DATA_BLOCK "DOOR_EXTRACTOR_DB"	// DB 12
AUTHOR : Kamillas
VERSION : 0.1
  STRUCT
   DOOR_EXT_LOC_SS : BOOL ;	//DOOR EXTRACTOR LOCAL SELECTOR SWITCH
   DOOR_EXT_MAN_SS : BOOL ;	//DOOR EXTRACTOR MANUAL SELECTOR SWITCH
   DOOR_EXT_AUTO_SS : BOOL ;	//DOOR EXTRACTOR AUTO SELECTOR SWITCH
   DOOR_EXT_STP_PB : BOOL ;	//DOOR EXTRACTOR STOP PUSH BUTTON
   SLEW_FWD_STA_PB : BOOL ;	//SLEW FORWARD START PUSH BUTTON
   SLEW_RET_STA_PB : BOOL ;	//SLEW RETRACT START
   VER_COMP_FWD_STA_PB : BOOL ;	//VERTICAL COMPENSATION FORWARD START PUSH BUTTON
   VER_COMP_RET_STA_PB : BOOL ;	//VERTICAL COMPENSATION RETRACT START PUSH BUTTON
   TRA_FWD_STA_PB : BOOL ;	//TRAVEL FORWARD START PUSH BUTTON
   TRA_RET_STA_PB : BOOL ;	//TRAVEL RETRACT START PUSH BUTTON
   MAIN_STK_UP_STA_PB : BOOL ;	//MAIN STROKE UP START PUSH BUTTON
   MAIN_STK_UP_DN_PB : BOOL ;	//MAIN STROKE DOWN START PUSH BUTTON
   FIN_STK_UP_STA_PB : BOOL ;	//FINAL STROKE UP START PUSH BUTTON
   FIN_STK_UP_DN_PB : BOOL ;	//FINAL STROKE DOWN START PUSH BUTTON
   PRE_STK_UP_STA_PB : BOOL ;	//PRE STROKE UP START PUSH BUTTON
   PRE_STK_UP_DN_PB : BOOL ;	//PRE STROKE DOWN START PUSH BUTTON
   DR_SPNG_LK_STA_PB : BOOL ;	//DOOR SPRING PRESSURE START PUSH BUTTON
   DR_SPNG_UNLK_STA_PB : BOOL ;	//DOOR SPRING PRESSURE RELEASE START PUSH BUTTON
   DR_LCH_TURN_UP_PB : BOOL ;	//DOOR LATCH TURNING LOCK PUSH BUTTON
   DR_LCH_TURN_DN_PB : BOOL ;	//DOOR LATCH TURNING UNLOCK PUSH BUTTON
   EMERGENCY_PB_LCS_73 : BOOL ;	//EMERGENCY PUSHBUTTON LCS-73
   SLEW_FWD_STA_PB_LCS : BOOL ;	//SLEW FORWARD START PUSH BUTTON LCS
   SLEW_RET_STA_PB_LCS : BOOL ;	//SLEW RETRACT START PUSHBUTTON LCS
   VER_COMP_FWD_STA_PB_LCS : BOOL ;	//VERTICAL COMPENSATION FORWARD START LCS PUSH BUTTON
   VER_COMP_RET_STA_PB_LCS : BOOL ;	//VERTICAL COMPENSATION RETRACT START LCS PUSH BUTTON
   TRA_FWD_STA_PB_LCS : BOOL ;	//TRAVEL FORWARD START LCS  PUSH BUTTON
   TRA_RET_STA_PB_LCS : BOOL ;	//TRAVEL BACK START LCS  PUSH BUTTON
   MAIN_STK_UP_STA_PB_LCS : BOOL ;	//MAIN STROKE UP START LCS PUSH BUTTON
   MAIN_STK_DN_STA_PB_LCS : BOOL ;	//MAIN STROKE DN START LCS PUSH BUTTON
   FIN_STK_UP_STA_PB_LCS : BOOL ;	//FINAL STROKE UP START LCS  PUSH BUTTON
   FIN_STK_DN_STA_PB_LCS : BOOL ;	//FINAL STROKE DOWN START LCS PUSH BUTTON
   PRE_STK_UP_STA_PB_LCS : BOOL ;	//PREE STROKE UP START LCS PUSH BUTTON
   PRE_STK_DN_STA_PB_LCS : BOOL ;	//PREE STROKE DN START LCS PUSH BUTTON
   DR_SPNG_LK_STA_PB_LCS : BOOL ;	//DOOR SPRING LOCK START PUSH BUTTON LCS
   DR_SPNG_UNLK_STA_PB_LCS : BOOL ;	//DOOR SPRING UNLOCK  START PUSH BUTTON LCS
   LAMP_TEST_PB_LCS_73 : BOOL ;	//LAMP TEST PUSHBUTTON LCS-73
   DR_LCH_TURN_UP_PB_LCS : BOOL ;	//DOOR LATCH LOCK PUSH BUTTON LCS
   DR_LCH_TURN_DN_PB_LCS : BOOL ;	//DOOR LATCH UNLOCK PUSH BUTTON LCS
   DR_LCH_TURN_HOME_PB_LCS : BOOL ;	//DOOR LATCH HOME PUSH BUTTON LCS
   SLEW_SLOW_FWD_LS : BOOL ;	//SLEW SLOW FORWARD LIMIT SWITCH
   SLEW_SLOW_RET_LS : BOOL ;	//SLEW SLOW RETRACT LIMIT SWITCH
   SLEW_NOR_FWD_LS : BOOL ;	//SLEW NORMAL FORWARD LIMIT SWITCH
   SLEW_NOR_RET_LS : BOOL ;	//SLEW NORMAL RETRACT LIMIT SWITCH
   TRA_SLOW_FWD_LS : BOOL ;	//TRAVEL SLOW FORWARD LIMIT  SWITCH
   TRA_SLOW_RET_LS : BOOL ;	//TRAVEL SLOW RETRACT LIMIT  SWITCH
   TRA_FWD_LS : BOOL ;	//TRAVEL FORWARD LIMIT SWIITCH
   TRA_RET_LS : BOOL ;	//TRAVEL RETRACT LIMIT SWIITCH
   FOR_LS_TRAVEL : BOOL ;	//FORWARD LIMIT SWITCH TRAVEL
   DOOR_ON_HOOK_LS : BOOL ;	//DOOR ON HOOK LIMITSWTCH
   DOOR_FIX_LOC_FB_PR_SWT : BOOL ;	//DOOR FIX LOCKED FEEDBACK PRESSURE SWITCH
   DR_LCH_TURN_UP_LS : BOOL ;	//DOOR LATCH TURNING UP LIMIT SWICH
   DR_LCH_TURN_DN_LS : BOOL ;	//DOOR LATCH TURNING DOWN LIMIT SWICH
   SPRING_PRESS : BOOL ;	//SPRING PRESS
   SLEW_SLOW_FWD_CMD : BOOL ;	//SLEW SLOW FORWARD COMMAND
   SLEW_SLOW_RET_CMD : BOOL ;	//SLEW SLOW RETRACT COMMAND
   SLEW_NOR_FWD_COMMAND : BOOL ;	//SLEW NORMAL FORWARD COMMAND
   SLEW_NOR_RET_COMMAND : BOOL ;	//SLEW NORMAL RETRACT COMMAND
   VER_COMP_FWD_CMD : BOOL ;	//VERTICAL COMPENSATION FORWARD COMMAND
   VER_COMP_RET_CMD : BOOL ;	//VERTICAL COMPENSATION RETRACT COMMAND
   VER_COMP_RELIVE_CMD : BOOL ;	//VERTICAL COMPENSTAION RELIVE  COOMMAND
   TRA_SLOW_FWD_CMD : BOOL ;	//TRAVEL SLOW FORWARD COMMAND
   TRA_SLOW_RET_CMD : BOOL ;	//TRAVEL SLOW RETRACT COMMAND
   TRA_NOR_FWD_CMD : BOOL ;	//TRAVEL NORMAL FORWARD COMMAND
   TRA_NOR_RET_CMD : BOOL ;	//TRAVEL NORMAL RETRACT COMMAND
   TRA_RELIVE_CMD : BOOL ;	//TRAVEL RELIVE COOMMAND
   MAIN_STK_UP_CMD : BOOL ;	//MANUAL STROKE UP COMMAND
   MAIN_STK_DN_CMD : BOOL ;	//MANUAL STROKE DN COMMAND
   PRE_STK_UP_CMD : BOOL ;	//PRE STROKE UP COMMAND
   PRE_STK_DN_CMD : BOOL ;	//PRE STROKE DN COMMAND
   DR_SPNG_LK_CMD : BOOL ;	//DOOR SPRING PRESS LOCK COMMAND
   DR_SPNG_UNLK_CMD : BOOL ;	//DOOR SPRING PRESS UNLOCK COMMAND
   DR_LCH_TURN_UP_CMD : BOOL ;	//DOOR LATCH TURNING UP COMMAND
   DR_LCH_TURN_DN_CMD : BOOL ;	//DOOR LATCH TURNING DOWN COMMADN
   SLEW_SLOW_FWD_IND : BOOL ;	//SLEW SLOW FORWARD INDICATOR
   SLEW_SLOW_RET_IND : BOOL ;	//SLEW SLOW RETRACT INDICATOR
   VER_COMP_FWD_IND : BOOL ;	//VERTICAL COMPENSATION FORWARD INDICATOR
   VER_COMP_RET_IND : BOOL ;	//VERTICAL COMPENSATION RETRACT INDICATOR
   TRA_FWD_IND : BOOL ;	//TRAVEL FORWARD INDICATOR
   TRA_RET_IND : BOOL ;	//TRAVEL BACK INDICATOR
   MAIN_STK_UP_IND : BOOL ;	//FINAL STROKE  UP INDICATION
   MAIN_STK_DN_IND : BOOL ;	//FINAL STROKE  DOWN  INDICATOR
   FIN_STK_UP_IND : BOOL ;	//FINAL STROKE  UP INDICATOR
   FIN_STK_DN_IND : BOOL ;	//FINAL STROKE  DOWN INDICATOR
   PRE_STK_UP_IND : BOOL ;	//PRE STROKE  UP INDICATION
   PRE_STK_DN_IND : BOOL ;	//PRE STROKE  DOWN INDICATOR
   DR_SPNG_LK_IND : BOOL ;	//DOOR SPRING PRESS LOCK INDICATOR
   DR_SPNG_UNLK_IND : BOOL ;	//DOOR SPRING PRESS UNLOCK INDICATOR
   DOOR_FIX_LOCK_IND : BOOL ;	//DOOR FIX LOCK INDICATOR
   DOOR_FIX_UNLK_IND : BOOL ;	//DOOR FIX UNLOCK INDICATOR
   DOOR_FIX_UNLK_IND1 : BOOL ;	//DOOR FIX UNLOCK INDICATOR
   LCS_73_ON_IND : BOOL ;	//LCS-73_ON_INDICATOR
   SLEW_SLOW_FWD_IND_LCS : BOOL ;	//SLEW SLOW FORWARD INDICATOR LCS
   SLEW_SLOW_RET_IND_LCS : BOOL ;	//SLEW SLOW RETRACT INDICATOR LCS
   VER_COMP_FWD_IND_LCS : BOOL ;	//VERTICAL COMPENSATION FORWARD INDICATOR LCS
   VER_COMP_RET_IND_LCS : BOOL ;	//VERTICAL COMPENSATION RETRACT INDICATOR LCS
   TRA_FWD_IND_LCS : BOOL ;	//TRAVEL FORWARD INDICATOR
   TRA_RET_IND_LCS : BOOL ;	//TRAVEL BACK INDICATOR LCS
   MAIN_STK_UP_IND_LCS : BOOL ;	//FINAL STROKE UP INDICATION LCS
   MAIN_STK_DN_IND_LCS : BOOL ;	//FINAL STROKE DOWN  INDICATOR LCS
   FIN_STK_UP_IND_LCS : BOOL ;	//FINAL STROKE UP INDICATOR LCS
   FIN_STK_DN_IND_LCS : BOOL ;	//FINAL STROKE DOWN INDICATOR LCS
   PRE_STK_UP_IND_LCS : BOOL ;	//PRE STROKE UP INDICATION LCS
   PRE_STK_DN_IND_LCS : BOOL ;	//PRE STROKE DOWN INDICATOR LCS
   DR_LCH_TURN_HOME_IND_LCS : BOOL ;	//DOOR LATCH HOME INDICATION LCS
   DR_LCH_TURN_UP_IND_LCS : BOOL ;	//DOOR LATCH TURNING UP INDICATOR LCS
   DR_LCH_TURN_DN_IND_LCS : BOOL ;	//DOOR LATCH TURNING DOWN INDICATOR LCS
   DOOR_FIX_LOCK_IND_LCS : BOOL ;	//DOOR FIX LOCK INDICATOR LCS
   DOOR_FIX_UNLK_IND_LCS : BOOL ;	//DOOR FIX UNLOCK INDICATOR LCS
   SLEW_SL_FWD_OP_CUT : BOOL ;	//SLEW SLOW FORWARD OUTPUT CUT
   SLEW_SL_FWD_FLT_TMR : INT ;	//SLEW SLOW FORWARD FAULT TIMER
   SLEW_SL_FWD_FLT_GEN : INT  := 8;	//SLEW SLOW FORWARD FAULT GENERATION TIME
   SLEW_SL_FWD_OP_CT_TM : INT ;	//SLEW SLOW FORWARD OUTPUT CUT TIMER
   SLEW_SL_FWD_FLT : BOOL ;	//SLEW SLOW FORWARD FAULT
   SLEW_SL_AUTO_FWD_OVR : BOOL ;	//SLEW SLOW AUTO FORWARD OVER
   SLEW_SL_AUTO_FWD_DEL : INT  := 3;	//SLEW SLOW AUTO FORWARD OVER DELAY
   SLEW_SL_ATO_FWD_DL_T : INT ;	//SLEW SLOW AUTO FORWARD OVER DELAY TIMER
   SLEW_NR_FWD_OP_CUT : BOOL ;	//SLEW NORMAL FORWARD OUTPUT CUT
   SLEW_NR_FWD_FLT_TMR : INT ;	//SLEW NORMAL FORWARD FAULT TIMER
   SLEW_NR_FWD_FLT_GEN : INT  := 8;	//SLEW NORMAL FORWARD FAULT GENERATION TIME
   SLEW_NR_FWD_OP_CT_TM : INT ;	//SLEW NORMAL FORWARD OUTPUT CUT TIMER
   SLEW_NR_FWD_FLT : BOOL ;	//SLEW NORMAL FORWARD FAULT
   SLEW_NR_AUTO_FWD_OVR : BOOL ;	//SLEW NORMAL AUTO FORWARD OVER
   SLEW_NR_AUTO_FWD_DEL : INT  := 3;	//SLEW NORMAL AUTO FORWARD OVER DELAY
   SLEW_NR_ATO_FWD_DL_T : INT ;	//SLEW NORMAL AUTO FORWARD OVER DELAY TIMER
   PULSE_1 : BOOL ;	//PULSE 1
   PULSE_2 : BOOL ;	//PULSE 2
   PULSE_3 : BOOL ;	//PULSE 3
   PULSE_4 : BOOL ;	//PULSE 4
   PULSE_5 : BOOL ;	//PULSE 5
   PULSE_6 : BOOL ;	//PULSE 6
   PULSE_7 : BOOL ;	//PULSE 7
   PULSE_8 : BOOL ;	//PULSE 8
   PULSE_9 : BOOL ;	//PULSE 9
   PULSE_10 : BOOL ;	//PULSE 10
   PULSE_11 : BOOL ;	//PULSE 11
   PULSE_12 : BOOL ;	//PULSE 12
   PULSE_13 : BOOL ;	//PULSE 13
   PULSE_14 : BOOL ;	//PULSE 14
   PULSE_15 : BOOL ;	//PULSE 15
   PULSE_16 : BOOL ;	//PULSE 16
   SLEW_NR_RET_OP_CUT : BOOL ;	//SLEW NORMAL RETRACT OUTPUT CUT
   SLEW_NR_RET_FLT_TMR : INT ;	//SLEW NORMAL RETRACT FAULT TIMER
   SLEW_NR_RET_FLT_GEN : INT  := 8;	//SLEW NORMAL RETRACT FAULT GENERATION TIME
   SLEW_NR_RET_OP_CT_TM : INT ;	//SLEW NORMAL RETRACT RETRACT OUTPUT CUT TIMER
   SLEW_NR_RET_FLT : BOOL ;	//SLEW NORMAL RETRACT RETRACT FAULT
   SLEW_NR_AUTO_RET_OVR : BOOL ;	//SLEW NORMAL AUTO RETRACT OVER
   SLEW_NR_AUTO_RET_DEL : INT  := 3;	//SLEW NORMAL AUTO RETRACT OVER DELAY
   SLEW_NR_ATO_RET_DL_T : INT ;	//SLEW NORMAL AUTO RETRACT OVER DELAY TIMER
   VER_COMP_FWD_OP_CUT : BOOL ;	//VERTICAL COMPENSATION FORWARD OUTPUT CUT
   VER_COMP_FWD_FLT_TMR : INT ;	//VERTICAL COMPENSATION FORWARD FAULT TIMER
   VER_COMP_FWD_FLT_GEN : INT  := 8;	//VERTICAL COMPENSATION FORWARD FAULT GENERATION TIME
   VER_COMP_FWD_OP_CT_TM : INT ;	//VERTICAL COMPENSATION FORWARD OUTPUT CUT TIMER
   VER_COMP_FWD_FLT : BOOL ;	//VERTICAL COMPENSATION FORWARD FAULT
   VER_COMP_AUTO_FWD_OVR : BOOL ;	//VERTICAL COMPENSATION AUTO FORWARD OVER
   VER_COMP_AUTO_FWD_DEL : INT  := 3;	//VERTICAL COMPENSATION AUTO FORWARD OVER DELAY
   VER_COMP_ATO_FWD_DL_T : INT ;	//VERTICAL COMPENSATION AUTO FORWARD OVER DELAY TIMER
   VER_COMP_RET_OP_CUT : BOOL ;	//VERTICAL COMPENSATION RETRACT OUTPUT CUT
   VER_COMP_RET_FLT_TMR : INT ;	//VERTICAL COMPENSATION RETRACT FAULT TIMER
   VER_COMP_RET_FLT_GEN : INT  := 8;	//VERTICAL COMPENSATION RETRACT FAULT GENERATION TIME
   VER_COMP_RET_OP_CT_TM : INT ;	//VERTICAL COMPENSATION RETRACT OUTPUT CUT TIMER
   VER_COMP_RET_FLT : BOOL ;	//VERTICAL COMPENSATION RETRACT FAULT
   VER_COMP_AUTO_RET_OVR : BOOL ;	//VERTICAL COMPENSATION AUTO RETRACT OVER
   VER_COMP_AUTO_RET_DEL : INT  := 3;	//VERTICAL COMPENSATION AUTO RETRACT OVER DELAY
   VER_COMP_ATO_RET_DL_T : INT ;	//VERTICAL COMPENSATION AUTO RETRACT OVER DELAY TIMER
   TRA_SLOW_FWD_OP_CUT : BOOL ;	//TRAVEL SLOW FORWARD OUTPUT CUT
   TRA_SLOW_FWD_FLT_TMR : INT ;	//TRAVEL SLOW FORWARD FAULT TIMER
   TRA_SLOW_FWD_FLT_GEN : INT  := 8;	//TRAVEL SLOW FORWARD FAULT GENERATION TIME
   TRA_SLOW_FWD_OP_CT_TM : INT ;	//TRAVEL SLOW FORWARD OUTPUT CUT TIMER
   TRA_SLOW_FWD_FLT : BOOL ;	//TRAVEL SLOW FORWARD FAULT
   TRA_SLOW_AUTO_FWD_OVR : BOOL ;	//TRAVEL SLOW AUTO FORWARD OVER
   TRA_SLOW_AUTO_FWD_DEL : INT  := 3;	//TRAVEL SLOW AUTO FORWARD OVER DELAY
   TRA_SLOW_ATO_FWD_DL_T : INT ;	//TRAVEL SLOW AUTO FORWARD OVER DELAY TIMER
   TRA_SLOW_RET_OP_CUT : BOOL ;	//TRAVEL SLOW RETRACT OUTPUT CUT
   TRA_SLOW_RET_FLT_TMR : INT ;	//TRAVEL SLOW RETRACT FAULT TIMER
   TRA_SLOW_RET_FLT_GEN : INT  := 8;	//TRAVEL SLOW RETRACT FAULT GENERATION TIME
   TRA_SLOW_RET_OP_CT_TM : INT ;	//TRAVEL SLOW RETRACT OUTPUT CUT TIMER
   TRA_SLOW_RET_FLT : BOOL ;	//TRAVEL SLOW RETRACT FAULT
   TRA_SLOW_AUTO_RET_OVR : BOOL ;	//TRAVEL SLOW AUTO RETRACT OVER
   TRA_SLOW_AUTO_RET_DEL : INT  := 3;	//TRAVEL SLOW AUTO RETRACT OVER DELAY
   TRA_SLOW_ATO_RET_DL_T : INT ;	//TRAVEL SLOW AUTO RETRACT OVER DELAY TIMER
   TRA_NOR_FWD_OP_CUT : BOOL ;	//TRAVEL NORMAL FORWARD OUTPUT CUT
   TRA_NOR_FWD_FLT_TMR : INT ;	//TRAVEL NORMAL FORWARD FAULT TIMER
   TRA_NOR_FWD_FLT_GEN : INT  := 8;	//TRAVEL NORMAL FORWARD FAULT GENERATION TIME
   TRA_NOR_FWD_OP_CT_TM : INT ;	//TRAVEL NORMAL FORWARD OUTPUT CUT TIMER
   TRA_NOR_FWD_FLT : BOOL ;	//TRAVEL NORMAL FORWARD FAULT
   TRA_NOR_AUTO_FWD_OVR : BOOL ;	//TRAVEL NORMAL AUTO FORWARD OVER
   TRA_NOR_AUTO_FWD_DEL : INT  := 3;	//TRAVEL NORMAL AUTO FORWARD OVER DELAY
   TRA_NOR_ATO_FWD_DL_T : INT ;	//TRAVEL NORMAL AUTO FORWARD OVER DELAY TIMER
   TRA_NOR_RET_OP_CUT : BOOL ;	//TRAVEL NORMAL RETRACT OUTPUT CUT
   TRA_NOR_RET_FLT_TMR : INT ;	//TRAVEL NORMAL RETRACT FAULT TIMER
   TRA_NOR_RET_FLT_GEN : INT  := 8;	//TRAVEL NORMAL RETRACT FAULT GENERATION TIME
   TRA_NOR_RET_OP_CT_TM : INT ;	//TRAVEL NORMAL RETRACT OUTPUT CUT TIMER
   TRA_NOR_RET_FLT : BOOL ;	//TRAVEL NORMAL RETRACT FAULT
   TRA_NOR_AUTO_RET_OVR : BOOL ;	//TRAVEL NORMAL AUTO RETRACT OVER
   TRA_NOR_AUTO_RET_DEL : INT  := 3;	//TRAVEL NORMAL AUTO RETRACT OVER DELAY
   TRA_NOR_ATO_RET_DL_T : INT ;	//TRAVEL NORMAL AUTO RETRACT OVER DELAY TIMER
   MAIN_STK_UP_OP_CUT : BOOL ;	//MAIN STROK UP OUTPUT CUT
   MAIN_STK_UP_FLT_TMR : INT ;	//MAIN STROK UP FAULT TIMER
   MAIN_STK_UP_FLT_GEN : INT  := 8;	//MAIN STROK UP FAULT GENERATION TIME
   MAIN_STK_UP_OP_CT_TM : INT ;	//MAIN STROK UP OUTPUT CUT TIMER
   MAIN_STK_UP_FLT : BOOL ;	//MAIN STROK UP FAULT
   MAIN_STK_AUTO_UP_OVR : BOOL ;	//MAIN STROK AUTO UP OVER
   MAIN_STK_AUTO_UP_DEL : INT  := 3;	//MAIN STROK AUTO UP OVER DELAY
   MAIN_STK_ATO_UP_DL_T : INT ;	//MAIN STROK AUTO UP OVER DELAY TIMER
   MAIN_STK_DN_OP_CUT : BOOL ;	//MAIN STROK DOWN OUTPUT CUT
   MAIN_STK_DN_FLT_TMR : INT ;	//MAIN STROK DOWN FAULT TIMER
   MAIN_STK_DN_FLT_GEN : INT  := 8;	//MAIN STROK DOWN FAULT GENERATION TIME
   MAIN_STK_DN_OP_CT_TM : INT ;	//MAIN STROK DOWN OUTPUT CUT TIMER
   MAIN_STK_DN_FLT : BOOL ;	//MAIN STROK DOWN FAULT
   MAIN_STK_AUTO_DN_OVR : BOOL ;	//MAIN STROK AUTO DOWN OVER
   MAIN_STK_AUTO_DN_DEL : INT  := 3;	//MAIN STROK AUTO DOWN OVER DELAY
   MAIN_STK_ATO_DN_DL_T : INT ;	//MAIN STROK AUTO DOWN OVER DELAY TIMER
   PRE_STK_UP_OP_CUT : BOOL ;	//PRE STROK UP OUTPUT CUT
   PRE_STK_UP_FLT_TMR : INT ;	//PRE STROK UP FAULT TIMER
   PRE_STK_UP_FLT_GEN : INT  := 8;	//PRE STROK UP FAULT GENERATION TIME
   PRE_STK_UP_OP_CT_TM : INT ;	//PRE STROK UP OUTPUT CUT TIMER
   PRE_STK_UP_FLT : BOOL ;	//PRE STROK UP FAULT
   PRE_STK_AUTO_UP_OVR : BOOL ;	//PRE STROK AUTO UP OVER
   PRE_STK_AUTO_UP_DEL : INT  := 3;	//PRE STROK AUTO UP OVER DELAY
   PRE_STK_ATO_UP_DL_T : INT ;	//PRE STROK AUTO UP OVER DELAY TIMER
   PRE_STK_DN_OP_CUT : BOOL ;	//PRE STROK DOWN OUTPUT CUT
   PRE_STK_DN_FLT_TMR : INT ;	//PRE STROK DOWN FAULT TIMER
   PRE_STK_DN_FLT_GEN : INT  := 8;	//PRE STROK DOWN FAULT GENERATION TIME
   PRE_STK_DN_OP_CT_TM : INT ;	//PRE STROK DOWN OUTPUT CUT TIMER
   PRE_STK_DN_FLT : BOOL ;	//PRE STROK DOWN FAULT
   PRE_STK_AUTO_DN_OVR : BOOL ;	//PRE STROK AUTO DOWN OVER
   PRE_STK_AUTO_DN_DEL : INT  := 3;	//PRE STROK AUTO DOWN OVER DELAY
   PRE_STK_ATO_DN_DL_T : INT ;	//PRE STROK AUTO DOWN OVER DELAY TIMER
   FIN_STK_UP_OP_CUT : BOOL ;	//FINAL STROK UP OUTPUT CUT
   FIN_STK_UP_FLT_TMR : INT ;	//FINAL STROK UP FAULT TIMER
   FIN_STK_UP_FLT_GEN : INT  := 8;	//FINAL STROK UP FAULT GENERATION TIME
   FIN_STK_UP_OP_CT_TM : INT ;	//FINAL STROK UP OUTPUT CUT TIMER
   FIN_STK_UP_FLT : BOOL ;	//FINAL STROK UP FAULT
   FIN_STK_AUTO_UP_OVR : BOOL ;	//FINAL STROK AUTO UP OVER
   FIN_STK_AUTO_UP_DEL : INT  := 3;	//FINAL STROK AUTO UP OVER DELAY
   FIN_STK_ATO_UP_DL_T : INT ;	//FINAL STROK AUTO UP OVER DELAY TIMER
   FIN_STK_DN_OP_CUT : BOOL ;	//FINAL STROK DOWN OUTPUT CUT
   FIN_STK_DN_FLT_TMR : INT ;	//FINAL STROK DOWN FAULT TIMER
   FIN_STK_DN_FLT_GEN : INT  := 8;	//FINAL STROK DOWN FAULT GENERATION TIME
   FIN_STK_DN_OP_CT_TM : INT ;	//FINAL STROK DOWN OUTPUT CUT TIMER
   FIN_STK_DN_FLT : BOOL ;	//FINAL STROK DOWN FAULT
   FIN_STK_AUTO_DN_OVR : BOOL ;	//FINAL STROK AUTO DOWN OVER
   FIN_STK_AUTO_DN_DEL : INT  := 3;	//FINAL STROK AUTO DOWN OVER DELAY
   FIN_STK_ATO_DN_DL_T : INT ;	//FINAL STROK AUTO DOWN OVER DELAY TIMER
   FIN_STK_UP_CMD : BOOL ;	//FINAL STROKE UP COMMAND
   FIN_STK_DN_CMD : BOOL ;	//FINAL STROKE DOWN COMMAND
   DR_SPNG_LK_OP_CUT : BOOL ;	//DOOR SPRING PRESSURE LOCK OUTPUT CUT
   DR_SPNG_LK_FLT_TMR : INT ;	//DOOR SPRING PRESSURE LOCK FAULT TIMER
   DR_SPNG_LK_FLT_GEN : INT  := 8;	//DOOR SPRING PRESSURE LOCK FAULT GENERATION TIME
   DR_SPNG_LK_OP_CT_TM : INT ;	//DOOR SPRING PRESSURE LOCK OUTPUT CUT TIMER
   DR_SPNG_LK_FLT : BOOL ;	//DOOR SPRING PRESSURE LOCK FAULT
   DR_SPNG_AUTO_LK_OVR : BOOL ;	//DOOR SPRING AUTO PRESSURE LOCK OVER
   DR_SPNG_AUTO_LK_DEL : INT  := 3;	//DOOR SPRING AUTO PRESSURE LOCK OVER DELAY
   DR_SPNG_ATO_LK_DL_T : INT ;	//DOOR SPRING AUTO PRESSURE LOCK OVER DELAY TIMER
   DR_SPNG_UNLK_OP_CUT : BOOL ;	//DOOR SPRING PRESSURE UNLOCK OUTPUT CUT
   DR_SPNG_UNLK_FLT_TMR : INT ;	//DOOR SPRING PRESSURE UNLOCK FAULT TIMER
   DR_SPNG_UNLK_FLT_GEN : INT  := 8;	//DOOR SPRING PRESSURE UNLOCK FAULT GENERATION TIME
   DR_SPNG_UNLK_OP_CT_TM : INT ;	//DOOR SPRING PRESSURE UNLOCK OUTPUT CUT TIMER
   DR_SPNG_UNLK_FLT : BOOL ;	//DOOR SPRING PRESSURE UNLOCK FAULT
   DR_SPNG_AUTO_UNLK_OVR : BOOL ;	//DOOR SPRING AUTO PRESSURE UNLOCK OVER
   DR_SPNG_AUTO_UNLK_DEL : INT  := 3;	//DOOR SPRING AUTO PRESSURE UNLOCK OVER DELAY
   DR_SPNG_ATO_UNLK_DL_T : INT ;	//DOOR SPRING AUTO PRESSURE UNLOCK OVER DELAY TIMER
   PULSE_17 : BOOL ;	//PULSE 17
   PULSE_18 : BOOL ;	//PULSE 18
   PULSE_19 : BOOL ;	//PULSE 19
   PULSE_20 : BOOL ;	//PULSE 20
   PULSE_21 : BOOL ;	//PULSE 21
   PULSE_22 : BOOL ;	//PULSE 22
   PULSE_23 : BOOL ;	//PULSE 23
   PULSE_24 : BOOL ;	//PULSE 24
   PULSE_25 : BOOL ;	//PULSE 25
   PULSE_26 : BOOL ;	//PULSE 26
   PULSE_27 : BOOL ;	//PULSE 27
   PULSE_28 : BOOL ;	//PULSE 28
   PULSE_29 : BOOL ;	//PULSE 29
   PULSE_30 : BOOL ;	//PULSE 30
   DR_LCH_UP_OP_CUT : BOOL ;	//DOOR LATCH UP OUTPUT CUT
   DR_LCH_UP_FLT_TMR : INT ;	//DOOR LATCH UP FAULT TIMER
   DR_LCH_UP_FLT_GEN : INT  := 8;	//DOOR LATCH UP FAULT GENERATION TIME
   DR_LCH_UP_OP_CT_TM : INT ;	//DOOR LATCH UP OUTPUT CUT TIMER
   DR_LCH_UP_FLT : BOOL ;	//DOOR LATCH UP FAULT
   DR_LCH_AUTO_UP_OVR : BOOL ;	//DOOR LATCH AUTO PRESSURE UP OVER
   DR_LCH_AUTO_UP_DEL : INT  := 3;	//DOOR LATCH AUTO PRESSURE UP OVER DELAY
   DR_LCH_ATO_UP_DL_T : INT ;	//DOOR LATCH AUTO PRESSURE UP OVER DELAY TIMER
   DR_LCH_DN_OP_CUT : BOOL ;	//DOOR LATCH DOWN OUTPUT CUT
   DR_LCH_DN_FLT_TMR : INT ;	//DOOR LATCH DOWN FAULT TIMER
   DR_LCH_DN_FLT_GEN : INT  := 8;	//DOOR LATCH DOWN FAULT GENERATION TIME
   DR_LCH_DN_OP_CT_TM : INT ;	//DOOR LATCH DOWN OUTPUT CUT TIMER
   DR_LCH_DN_FLT : BOOL ;	//DOOR LATCH DOWN FAULT
   DR_LCH_AUTO_DN_OVR : BOOL ;	//DOOR SPRING AUTO PRESSURE DOWN OVER
   DR_LCH_AUTO_DN_DEL : INT  := 3;	//DOOR SPRING AUTO PRESSURE DOWN OVER DELAY
   DR_LCH_ATO_DN_DL_T : INT ;	//DOOR SPRING AUTO PRESSURE DOWN OVER DELAY TIMER
   TRA_SLOW_FWD_IND : BOOL ;	//TRAVEL SLOW FORWARD INDICATOR
   TRA_SLOW_RET_IND : BOOL ;	//TRAVEL SLOW RETRACT INDICATOR
   TRA_SLOW_FWD_IND_LCS : BOOL ;	//TRAVEL SLOW FORWARD INDICATOR LCS
   TRA_SLOW_RET_IND_LCS : BOOL ;	//TRAVEL RETRACT INDICATOR LCS
   SLEW_FWD_IND : BOOL ;	//SLEW NORMAL FORWARD INDICATOR
   SLEW_RET_IND : BOOL ;	//SLEW NORMAL RETRACT INDICATOR
   SLEW_FWD_IND_LCS : BOOL ;	//SLEW NORMAL FORWARD INDICATOR LCS
   SLEW_RET_IND_LCS : BOOL ;	//SLEW NORMAL RETRACT INDICATOR LCS
   DR_SPNG_LK_IND_LCS : BOOL ;	//DOOR SPRING PRESS LOCK INDICATOR LCS
   DR_SPNG_UNLK_IND_LCS : BOOL ;	//DOOR SPRING PRESS UNLOCK INDICATOR LCS
   DE_TRA_SLOW_FWD_BIT : BOOL ;	//DOOR EXTRACTOR TRAVEL SLOW FORWARD START BIT
   DOR_EXT_RPL_ILK_BIT : BOOL ;	//DOOR EXTRACTOR/REPLACE INTERLOCK BIT
   DR_EXT_AUTO_STA_BIT : BOOL ;	//DOOR EXTRACTOR AUTO START BIT
   EXT_OVEN_DOR_AUTO_STA_PB : BOOL ;	//EXTRACT OVEN DOOR AUTO START PUSH BUTTON
   DR_EXT_RPL_AUTO_STP_PB : BOOL ;	//DOOR EXTRACTOR/REPLACE AUTO STOP PUSH BUTTON
   RPL_OVEN_DOR_AUTO_STA_PB : BOOL ;	//REPLACE OVEN DOOR AUTO START PUSH BUTTON
   VER_COMP_LDT_SCLD_VLU : REAL ;	//VERTICAL COMPENSATION LDT SCALED VALUE
   VER_COMP_LDT_SLNG_ERR : WORD ;	//VERTICAL COMPENSATION LDT SCALING ERROR
   DR_RPL_AUTO_STA_BIT : BOOL ;	//DOOR REPLACE AUTO START BIT
   PULSE_31 : BOOL ;	//PULSE 31
   PULSE_32 : BOOL ;	//PULSE 32
   PULSE_33 : BOOL ;	//PULSE 33
   PULSE_34 : BOOL ;	//PULSE 34
   PULSE_35 : BOOL ;	//PULSE 35
   PULSE_36 : BOOL ;	//PULSE 36
   PULSE_37 : BOOL ;	//PULSE 37
   PULSE_38 : BOOL ;	//PULSE 38
   PULSE_39 : BOOL ;	//PULSE 39
   PULSE_40 : BOOL ;	//PULSE 40
   PULSE_41 : BOOL ;	//PULSE 41
   PULSE_42 : BOOL ;	//PULSE 42
   PULSE_43 : BOOL ;	//PULSE 43
   PULSE_44 : BOOL ;	//PULSE 44
   PULSE_45 : BOOL ;	//PULSE 45
   PULSE_46 : BOOL ;	//PULSE 46
   PULSE_47 : BOOL ;	//PULSE 47
   PULSE_48 : BOOL ;	//PULSE 48
   PULSE_49 : BOOL ;	//PULSE 49
   PULSE_50 : BOOL ;	//PULSE 50
   PRE_STK_UP_LR : BOOL ;	//PRE STROKE UP LIMIT READHED
   PRE_STK_DN_LR : BOOL ;	//PRE STROKE DOWN LIMIT READHED
   MAIN_STK_FWD_LR : BOOL ;	//MAIN STROKE UP LIMIT READHED
   MAIN_STK_DN_LR : BOOL ;	//MAIN STROKE DOWN LIMIT READHED
   FIN_STK_FWD_LR : BOOL ;	//FINAL STROKE UP LIMIT READHED
   FIN_STK_DN_LR : BOOL ;	//FINAL STROKE DOWN LIMIT READHED
   EXT_OVEN_DOR_IND : BOOL ;	//EEXTRACT OVEN DOOR INDICATOR
   RPL_OVEN_DOR_IND : BOOL ;	//REPLACE OVEN DOOR INDICATOR
   SLEW_AUTO_FWD_SET : BOOL ;	//SLWE AUTO FORWARD SET
   SLEW_AUTO_RET_SET : BOOL ;	//SLWE AUTO RETRACT SET
   VER_COMP_AUTO_FWD_SET : BOOL ;	//VERTICAL COMPENSATION AUTO FORWARD SET
   VER_COMP_AUTO_RET_SET : BOOL ;	//VERTICAL COMPENSATION AUTO RETRACT SET
   TRA_AUTO_FWD_SET : BOOL ;	//TRAVEL AUTO FORWARD SET
   TRA_AUTO_RET_SET : BOOL ;	//TRAVEL AUTO RETRACT SET
   PRE_STK_AUTO_FWD_SET : BOOL ;	//PRE STROK AUTO FORWARD SET
   PRE_STK_AUTO_RET_SET : BOOL ;	//PRE STROK AUTO RETRACT SET
   MAIN_STK_AUTO_FWD_SET : BOOL ;	//MAIN STROK AUTO FORWARD SET
   MAIN_STK_AUTO_RET_SET : BOOL ;	//MAIN STROK AUTO RETRACT SET
   FIN_STK_AUTO_FWD_SET : BOOL ;	//FINAL STROK AUTO FORWARD SET
   FIN_STK_AUTO_RET_SET : BOOL ;	//FINAL STROK AUTO RETRACT SET
   DR_SPNG_AUTO_PRSD_SET : BOOL ;	//DOOR SPING AUTO PRESSED SET
   DR_SRNG_AUTO_RLSD_SET : BOOL ;	//DOOR SPING AUTO RELESED SET
   DR_LCH_TURN_AUTO_UP_SET : BOOL ;	//DOOR LATCH TURN AUTO UP BIT
   DR_LCH_TURN_AUTO_DN_SET : BOOL ;	//DOOR LATCH TURN AUTO DOWN BIT
   DR_LFT_LDT_SCLD_VLU : REAL ;	//DOOR LIFTING LDT SCALED VALUE
   DR_LFT_LDT_SLNG_ERR : WORD ;	//DOOR LIFTING LDT SCALING ERROR
   VER_COMP_VALUE : REAL ;	//VERTICAL COMPENSATION VALUE
   VER_COMP_LDT_REAL : REAL ;	//VERTICAL COMPENSATION LDT REAL VALUE
   DR_LFT_LDT_REAL : REAL ;	//DOOR LIFTING LDT REAL VALUE
   VER_COMP_UNSCLD_VLU : INT ;	//VERTICAL COMPENSATION UNSCALED VALUE
   DR_LFT_UNSCLD_VLU : INT ;	//DOOR LIFTER UNSCALED VALUE
   PRE_STK_UP_LDT_VLU : REAL ;	//PRE STROKE UP LDT VALUE
   MAIN_STK_UP_LDT_VLU : REAL ;	//MAIN STROKE UP LDT VALUE
   FIN_STK_UP_LDT_VLU : REAL ;	//FIN STROKE UP LDT VALUE
   PRE_STK_DN_LDT_VLU : REAL ;	//PRE STROKE DOWN LDT VALUE
   MAIN_STK_DN_LDT_VLU : REAL ;	//MAIN STROKE DOWN LDT VALUE
   FIN_STK_DN_LDT_VLU : REAL ;	//FIN STROKE DOWN LDT VALUE
   VER_COMP_FWD_LIM_VALUE : REAL ;	//VERTICAL COMPENSATION FORWARD LIMIT VALUE
   DOOR_FIX_REL_FB : BOOL ;	//DOOR RELEASE FEEDBACK
   DR_LCH_TURN_UP_IND : BOOL ;	//DOOR LATCH LOCK INDICATOR CD
   DR_LCH_TURN_DN_IND : BOOL ;	//DOOR LATCH UNLOCK INDICATOR CD
   VER_COMP_LR : BOOL ;	//VERTICAL COMPENSATION LIMIT REACHED
   DR_EXTR_HME_POS : BOOL ;	//DOOR EXTRACTOR HOME POSITION REACHED
   DR_EXT_AUTO_OPER_FIN : BOOL ;	//DOOR EXTRACTOR AUTO OPERATIONS FINISHED
   DR_RPL_AUTO_OPER_FIN : BOOL ;	//DOOR REPLACE AUTO OPERATIONS FINISHED
   TRA_RELEVE_VLV : BOOL ;	//TRAVEL RELEVE VALVE
   VER_COMP_RELEVE_VLV : BOOL ;	//VERTICAL COMPENSATION RELEVE VALVE
   LIFT_LDT_TMR_SS : BOOL ;	//LIFTING CYLINDER LDT TIMER SELECTOR SWITCH
   PRE_STK_UP_TIM_OP_CUT : BOOL ;	//PRE STROKE UP TIMER OP CUT
   PRE_STK_DN_TIM_OP_CUT : BOOL ;	//PRE STROKE DOWN TIMER OP CUT
   MAIN_STK_UP_TIM_OP_CUT : BOOL ;	//MAIN STROKE UP TIMER OP CUT
   MAIN_STK_DN_TIM_OP_CUT : BOOL ;	//MAIN STROKE DOWN TIMER OP CUT
   FIN_STK_UP_TIM_OP_CUT : BOOL ;	//FINAL STROKE UP TIMER OP CUT
   FIN_STK_DN_TIM_OP_CUT : BOOL ;	//FINAL STROKE DOWN TIMER OP CUT
   SPARE : BOOL ;	//SPARE
   VERT_COMP_FWD_TIM_OP_CUT : BOOL ;	//VERTICAL COMPENSATION FORWARD OP CUT THRU TIMER
   VERT_COMP_RET_TIM_OP_CUT : BOOL ;	//VERTICAL COMPENSATION RETRACT OP CUT THRU TIMER
  END_STRUCT ;	
BEGIN
   SLEW_SL_FWD_FLT_GEN := 8;
   SLEW_SL_AUTO_FWD_DEL := 3;
   SLEW_NR_FWD_FLT_GEN := 8;
   SLEW_NR_AUTO_FWD_DEL := 3;
   SLEW_NR_RET_FLT_GEN := 8;
   SLEW_NR_AUTO_RET_DEL := 3;
   VER_COMP_FWD_FLT_GEN := 8;
   VER_COMP_AUTO_FWD_DEL := 3;
   VER_COMP_RET_FLT_GEN := 8;
   VER_COMP_AUTO_RET_DEL := 3;
   TRA_SLOW_FWD_FLT_GEN := 8;
   TRA_SLOW_AUTO_FWD_DEL := 3;
   TRA_SLOW_RET_FLT_GEN := 8;
   TRA_SLOW_AUTO_RET_DEL := 3;
   TRA_NOR_FWD_FLT_GEN := 8;
   TRA_NOR_AUTO_FWD_DEL := 3;
   TRA_NOR_RET_FLT_GEN := 8;
   TRA_NOR_AUTO_RET_DEL := 3;
   MAIN_STK_UP_FLT_GEN := 8;
   MAIN_STK_AUTO_UP_DEL := 3;
   MAIN_STK_DN_FLT_GEN := 8;
   MAIN_STK_AUTO_DN_DEL := 3;
   PRE_STK_UP_FLT_GEN := 8;
   PRE_STK_AUTO_UP_DEL := 3;
   PRE_STK_DN_FLT_GEN := 8;
   PRE_STK_AUTO_DN_DEL := 3;
   FIN_STK_UP_FLT_GEN := 8;
   FIN_STK_AUTO_UP_DEL := 3;
   FIN_STK_DN_FLT_GEN := 8;
   FIN_STK_AUTO_DN_DEL := 3;
   DR_SPNG_LK_FLT_GEN := 8;
   DR_SPNG_AUTO_LK_DEL := 3;
   DR_SPNG_UNLK_FLT_GEN := 8;
   DR_SPNG_AUTO_UNLK_DEL := 3;
   DR_LCH_UP_FLT_GEN := 8;
   DR_LCH_AUTO_UP_DEL := 3;
   DR_LCH_DN_FLT_GEN := 8;
   DR_LCH_AUTO_DN_DEL := 3;
END_DATA_BLOCK

DATA_BLOCK "DOOR_CLEANER_DB"	// DB 13
AUTHOR : Kamillas
VERSION : 0.1
  STRUCT
   DOOR_CLNR_LOC_SS : BOOL ;	//DOOR CLEANER LOCAL SELECTOR SWITCH
   DOOR_CLNR_MAN_SS : BOOL ;	//DOOR CLEANER MANUAL SELECTOR SWITCH
   DOOR_CLNR_AUTO_SS : BOOL ;	//DOOR CLEANER AUTO SELECTOR SWITCH
   DOOR_CLNR_STP_PB : BOOL ;	//DOOR CLEANER STOP PUSH BUTTON
   CAR_TRA_FWD_STA_PB : BOOL ;	//CARRIAGE TRAVEL FORWARD START PUSH BUTTON
   CAR_TRA_RET_STA_PB : BOOL ;	//CARRIAGE TRAVEL RETRACT START PUSH BUTTON
   VER_CLNR_UP_STA_PB : BOOL ;	//VERTICAL CLEANER UP START PUSH BUTTON
   VER_CLNR_DN_STA_PB : BOOL ;	//VERTICAL CLEANER DOWN START PUSH BUTTON
   BTM_BRK_HLDR_UP_STA_PB : BOOL ;	//BOTTOM BRICK HOLDER FORWARD START PUSH BUTTON
   BTM_BRK_HLDR_DN_STA_PB : BOOL ;	//BOTTOM BRICK HOLDER RETRACT START PUSH BUTTON
   TOP_SCRP_FWD_STA_PB : BOOL ;	//TOP SCRAPPER FORWARD START PUSH BUTTON
   TOP_SCRP_RET_STA_PB : BOOL ;	//TOP SCRAPPER RETRACT START PUSH BUTTON
   BTM_SCRP_FWD_STA_PB : BOOL ;	//BOTTOM SCRAPPER FORWARD START PUSH BUTTON
   BTM_SCRP_RET_STA_PB : BOOL ;	//BOTTOM SCRAPPER RETRACT START PUSH BUTTON
   EMERGENCY_STOP_PB_LCS_85 : BOOL ;	//EMERGENCY STOP PUSH BUTTON LCS 85
   CAR_TRA_FWD_STA_PB_LCS : BOOL ;	//CARRIAGE TRAVEL FORWARD START PUSH BUTTON LCS
   CAR_TRA_RET_STA_PB_LCS : BOOL ;	//CARRIAGE TRAVEL RETRACT START PUSH BUTTON LCS
   VER_CLNR_UP_STA_PB_LCS : BOOL ;	//VERTICAL CLEANER UP START PUSH BUTTON LCS
   VER_CLNR_DN_STA_PB_LCS : BOOL ;	//VERTICAL CLEANER DOWN START PUSH BUTTON LCS
   BTM_BRK_HLDR_UP_STA_LCS : BOOL ;	//BOTTOM BRICK HOLDER FORWARD START PUSH BUTTON LCS
   BTM_BRK_HLDR_DN_STA_LCS : BOOL ;	//BOTTOM BRICK HOLDER RETRACT START PUSH BUTTON LCS
   LAMP_TEST_PB_LCS_85 : BOOL ;	//LAMP TEST PUSH BUTTON LCS 85
   GRV_SCRP_FWD_PB_LCS : BOOL ;	//GROOVE SCRAPPER FWD PUSH BUTTON LCS
   GEV_SCRP_RET_PB_LCS : BOOL ;	//GROOVE SCRAPPER RETRACT PUSH BUTTON LCS
   TOP_SCRP_FWD_STA_PB_LCS : BOOL ;	//TOP SCRAPPER FORWARD START PUSH BUTTON LCS
   TOP_SCRP_RET_STA_PB_LCS : BOOL ;	//TOP SCRAPPER RETRACT START PUSH BUTTON LCS
   BTM_SCRP_FWD_STA_PB_LCS : BOOL ;	//BOTTOM SCRAPPER FORWARD START PUSH BUTTON LCS
   BTM_SCRP_RET_STA_PB_LCS : BOOL ;	//BOTTOM SCRAPPER RETRACT START PUSH BUTTON LCS
   CAR_TRA_FWD_LS : BOOL ;	//CARRIAGE TRAVEL FORWARD LIMIT SWITCH
   CAR_TRA_RET_LS : BOOL ;	//CARRIAGE TRAVEL RETRACT LIMIT SWITCH
   VER_CLNR_UP_LS : BOOL ;	//VERTICAL CLEANER UP START LIMIT SWITCH
   VER_CLNR_DN_LS : BOOL ;	//VERTICAL CLEANER DOWN START LIMIT SWITCH
   BTM_BRK_HLDR_UP_LS : BOOL ;	//BOTTOM BRICK HOLDER FORWARD LIMIT SWITCH
   BTM_BRK_HLDR_DN_LS : BOOL ;	//BOTTOM BRICK HOLDER RETRACT LIMIT SWITCH
   TOP_SCRP_FWD_LS : BOOL ;	//TOP SCRAPPER FORWARD LIMIT SWITCH
   TOP_SCRP_RET_LS : BOOL ;	//TOP SCRAPPER RETRACT LIMIT SWITCH
   BTM_SCRP_FWD_LS : BOOL ;	//BOTTOM SCRAPPER FORWARD LIMIT SWITCH
   BTM_SCRP_RET_LS : BOOL ;	//BOTTOM SCRAPPER RETRACT LIMIT SWITCH
   CAR_TRA_FWD_CMD : BOOL ;	//CARRIAGE TRAVEL FORWARD COMMAND
   CAR_TRA_RET_CMD : BOOL ;	//CARRIAGE TRAVEL RETRACT COMMAND
   VER_CLNR_UP_CMD : BOOL ;	//VERTICAL CLEANER UP START COMMAND
   VER_CLNR_DN_CMD : BOOL ;	//VERTICAL CLEANER DOWN START COMMAND
   BTM_BRK_HLDR_UP_CMD : BOOL ;	//BOTTOM BRICK HOLDER FORWARD COMMAND
   BTM_BRK_HLDR_DN_CMD : BOOL ;	//BOTTOM BRICK HOLDER RETRACT COMMAND
   TOP_SCRP_FWD_CMD : BOOL ;	//TOP SCRAPPER FORWARD COMMAND
   TOP_SCRP_RET_CMD : BOOL ;	//TOP SCRAPPER RETRACT COMMAND
   BTM_SCRP_FWD_CMD : BOOL ;	//BOTTOM SCRAPPER FORWARD COMMAND
   BTM_SCRP_RET_CMD : BOOL ;	//BOTTOM SCRAPPER RETRACT COMMAND
   CAR_TRA_FWD_IND : BOOL ;	//CARRIAGE TRAVEL FORWARD INDICATOR
   CAR_TRA_RET_IND : BOOL ;	//CARRIAGE TRAVEL RETRACT INDICATOR
   VER_CLNR_UP_IND : BOOL ;	//VERTICAL CLEANER UP START INDICATOR
   VER_CLNR_DN_IND : BOOL ;	//VERTICAL CLEANER DOWN START INDICATOR
   BTM_BRK_HLDR_UP_IND : BOOL ;	//BOTTOM BRICK HOLDER FORWARD INDICATOR
   BTM_BRK_HLDR_DN_IND : BOOL ;	//BOTTOM BRICK HOLDER RETRACT INDICATOR
   TOP_SCRP_FWD_IND : BOOL ;	//TOP SCRAPPER FORWARD INDICATOR
   TOP_SCRP_RET_IND : BOOL ;	//TOP SCRAPPER RETRACT INDICATOR
   BTM_SCRP_FWD_IND : BOOL ;	//BOTTOM SCRAPPER FORWARD INDICATOR
   BTM_SCRP_RET_IND : BOOL ;	//BOTTOM SCRAPPER RETRACT INDICATOR
   CAR_TRA_FWD_IND_LCS : BOOL ;	//CARRIAGE TRAVEL FORWARD INDICATOR LCS
   CAR_TRA_RET_IND_LCS : BOOL ;	//CARRIAGE TRAVEL RETRACT INDICATOR LCS
   VER_CLNR_UP_IND_LCS : BOOL ;	//VERTICAL CLEANER UP START INDICATOR LCS
   VER_CLNR_DN_IND_LCS : BOOL ;	//VERTICAL CLEANER DOWN START INDICATOR LCS
   BTM_BRK_HLDR_UP_IND_LCS : BOOL ;	//BOTTOM BRICK HOLDER FORWARD INDICATOR LCS
   BTM_BRK_HLDR_DN_IND_LCS : BOOL ;	//BOTTOM BRICK HOLDER RETRACT INDICATOR LCS
   TOP_SCRP_FWD_IND_LCS : BOOL ;	//TOP SCRAPPER FORWARD INDICATOR LCS
   TOP_SCRP_RET_IND_LCS : BOOL ;	//TOP SCRAPPER RETRACT INDICATOR LCS
   BTM_SCRP_FWD_IND_LCS : BOOL ;	//BOTTOM SCRAPPER FORWARD INDICATOR LCS
   BTM_SCRP_RET_IND_LCS : BOOL ;	//BOTTOM SCRAPPER RETRACT INDICATOR LCS
   LCS_85_0N_IND : BOOL ;	//LCS-85 ON INDICATOR
   GRV_SRPR_FWD_IND_LCS : BOOL ;	//GROOVE SCRAPPER FORWARD INDICATOR LCS
   GRV_SRPR_RET_IND_LCS : BOOL ;	//GROOVE SCRAPPER RETRACT INDICATOR LCS
   CAR_TRA_FWD_OP_CUT : BOOL ;	//CARRIAGE TRAVEL FORWARD OUTPUT CUT
   CAR_TRA_FWD_FLT_TMR : INT ;	//CARRIAGE TRAVEL FORWARD FAULT TIMER
   CAR_TRA_FWD_FLT_GEN : INT  := 8;	//CARRIAGE TRAVEL FORWARD FAULT GENERATION TIME
   CAR_TRA_FWD_OP_CT_TM : INT ;	//CARRIAGE TRAVEL FORWARD OUTPUT CUT TIMER
   CAR_TRA_FWD_FLT : BOOL ;	//CARRIAGE TRAVEL FORWARD FAULT
   CAR_TRA_AUTO_FWD_OVR : BOOL ;	//CARRIAGE TRAVEL AUTO FORWARD OVER
   CAR_TRA_AUTO_FWD_DEL : INT  := 3;	//CARRIAGE TRAVEL AUTO FORWARD OVER DELAY
   CAR_TRA_ATO_FWD_DL_T : INT ;	//CARRIAGE TRAVEL AUTO FORWARD OVER DELAY TIMER
   PULSE_1 : BOOL ;	//PULSE 1
   PULSE_2 : BOOL ;	//PULSE 2
   PULSE_3 : BOOL ;	//PULSE 3
   PULSE_4 : BOOL ;	//PULSE 4
   PULSE_5 : BOOL ;	//PULSE 5
   PULSE_6 : BOOL ;	//PULSE 6
   PULSE_7 : BOOL ;	//PULSE 7
   PULSE_8 : BOOL ;	//PULSE 8
   PULSE_9 : BOOL ;	//PULSE 9
   PULSE_10 : BOOL ;	//PULSE 10
   PULSE_11 : BOOL ;	//PULSE 11
   PULSE_12 : BOOL ;	//PULSE 12
   PULSE_13 : BOOL ;	//PULSE 13
   PULSE_14 : BOOL ;	//PULSE 14
   PULSE_15 : BOOL ;	//PULSE 15
   PULSE_16 : BOOL ;	//PULSE 16
   CAR_TRA_RET_OP_CUT : BOOL ;	//CARRIAGE TRAVEL RETRACT OUTPUT CUT
   CAR_TRA_RET_FLT_TMR : INT ;	//CARRIAGE TRAVEL RETRACT FAULT TIMER
   CAR_TRA_RET_FLT_GEN : INT  := 8;	//CARRIAGE TRAVEL RETRACT FAULT GENERATION TIME
   CAR_TRA_RET_OP_CT_TM : INT ;	//CARRIAGE TRAVEL RETRACT OUTPUT CUT TIMER
   CAR_TRA_RET_FLT : BOOL ;	//CARRIAGE TRAVEL RETRACT FAULT
   CAR_TRA_AUTO_RET_OVR : BOOL ;	//CARRIAGE TRAVEL AUTO RETRACT OVER
   CAR_TRA_AUTO_RET_DEL : INT  := 3;	//CARRIAGE TRAVEL AUTO RETRACT OVER DELAY
   CAR_TRA_ATO_RET_DL_T : INT ;	//CARRIAGE TRAVEL AUTO RETRACT OVER DELAY TIMER
   VER_CLNR_UP_OP_CUT : BOOL ;	//VERTICAL CLEANER UP OUTPUT CUT
   VER_CLNR_UP_FLT_TMR : INT ;	//VERTICAL CLEANER UP FAULT TIMER
   VER_CLNR_UP_FLT_GEN : INT  := 8;	//VERTICAL CLEANER UP FAULT GENERATION TIME
   VER_CLNR_UP_OP_CT_TM : INT ;	//VERTICAL CLEANER UP OUTPUT CUT TIMER
   VER_CLNR_UP_FLT : BOOL ;	//VERTICAL CLEANER UP FAULT
   VER_CLNR_AUTO_UP_OVR : BOOL ;	//VERTICAL CLEANER AUTO UP OVER
   VER_CLNR_AUTO_UP_DEL : INT  := 3;	//VERTICAL CLEANER AUTO UP OVER DELAY
   VER_CLNR_ATO_UP_DL_T : INT ;	//VERTICAL CLEANER AUTO UP OVER DELAY TIMER
   VER_CLNR_DN_OP_CUT : BOOL ;	//VERTICAL CLEANER DOWN OUTPUT CUT
   VER_CLNR_DN_FLT_TMR : INT ;	//VERTICAL CLEANER DOWN FAULT TIMER
   VER_CLNR_DN_FLT_GEN : INT  := 8;	//VERTICAL CLEANER DOWN FAULT GENERATION TIME
   VER_CLNR_DN_OP_CT_TM : INT ;	//VERTICAL CLEANER DOWN OUTPUT CUT TIMER
   VER_CLNR_DN_FLT : BOOL ;	//VERTICAL CLEANER DOWN FAULT
   VER_CLNR_AUTO_DN_OVR : BOOL ;	//VERTICAL CLEANER AUTO DOWN OVER
   VER_CLNR_AUTO_DN_DEL : INT  := 3;	//VERTICAL CLEANER AUTO DOWN OVER DELAY
   VER_CLNR_ATO_DN_DL_T : INT ;	//VERTICAL CLEANER AUTO DOWN OVER DELAY TIMER
   BTM_BRK_HLDR_DN_OP_CUT : BOOL ;	//BOTTOM BRICK HOLDER DOWN OUTPUT CUT
   BTM_BRK_HLDR_DN_FLT_TMR : INT ;	//BOTTOM BRICK HOLDER DOWN FAULT TIMER
   BTM_BRK_HLDR_DN_FLT_GEN : INT  := 8;	//BOTTOM BRICK HOLDER DOWN FAULT GENERATION TIME
   BTM_BRK_HLDR_DN_OP_CT_TM : INT ;	//BOTTOM BRICK HOLDER DOWN OUTPUT CUT TIMER
   BTM_BRK_HLDR_DN_FLT : BOOL ;	//BOTTOM BRICK HOLDER DOWN FAULT
   BTM_BRK_HLDR_AUTO_DN_OVR : BOOL ;	//BOTTOM BRICK HOLDER AUTO DOWN OVER
   BTM_BRK_HLDR_AUTO_DN_DEL : INT  := 3;	//BOTTOM BRICK HOLDER AUTO DOWN OVER DELAY
   BTM_BRK_HLDR_ATO_DN_DL_T : INT ;	//BOTTOM BRICK HOLDER AUTO DOWN OVER DELAY TIMER
   BTM_BRK_HLDR_UP_OP_CUT : BOOL ;	//BOTTOM BRICK HOLDER UP OUTPUT CUT
   BTM_BRK_HLDR_UP_FLT_TMR : INT ;	//BOTTOM BRICK HOLDER UP FAULT TIMER
   BTM_BRK_HLDR_UP_FLT_GEN : INT  := 8;	//BOTTOM BRICK HOLDER UP FAULT GENERATION TIME
   BTM_BRK_HLDR_UP_OP_CT_TM : INT ;	//BOTTOM BRICK HOLDER UP OUTPUT CUT TIMER
   BTM_BRK_HLDR_UP_FLT : BOOL ;	//BOTTOM BRICK HOLDER UP FAULT
   BTM_BRK_HLDR_AUTO_UP_OVR : BOOL ;	//BOTTOM BRICK HOLDER AUTO UP OVER
   BTM_BRK_HLDR_AUTO_UP_DEL : INT  := 3;	//BOTTOM BRICK HOLDER AUTO UP OVER DELAY
   BTM_BRK_HLDR_ATO_UP_DL_T : INT ;	//BOTTOM BRICK HOLDER AUTO UP OVER DELAY TIMER
   TOP_SCRP_FWD_OP_CUT : BOOL ;	//TOP SCRAPPER FORWARD OUTPUT CUT
   TOP_SCRP_FWD_FLT_TMR : INT ;	//TOP SCRAPPER FORWARD FAULT TIMER
   TOP_SCRP_FWD_FLT_GEN : INT  := 8;	//TOP SCRAPPER FORWARD FAULT GENERATION TIME
   TOP_SCRP_FWD_OP_CT_TM : INT ;	//TOP SCRAPPER FORWARD OUTPUT CUT TIMER
   TOP_SCRP_FWD_FLT : BOOL ;	//TOP SCRAPPER FORWARD FAULT
   TOP_SCRP_AUTO_FWD_OVR : BOOL ;	//TOP SCRAPPER AUTO FORWARD OVER
   TOP_SCRP_AUTO_FWD_DEL : INT  := 3;	//TOP SCRAPPER AUTO FORWARD OVER DELAY
   TOP_SCRP_ATO_FWD_DL_T : INT ;	//TOP SCRAPPER AUTO FORWARD OVER DELAY TIMER
   TOP_SCRP_RET_OP_CUT : BOOL ;	//TOP SCRAPPER RETRACT OUTPUT CUT
   TOP_SCRP_RET_FLT_TMR : INT ;	//TOP SCRAPPER RETRACT FAULT TIMER
   TOP_SCRP_RET_FLT_GEN : INT  := 8;	//TOP SCRAPPER RETRACT FAULT GENERATION TIME
   TOP_SCRP_RET_OP_CT_TM : INT ;	//TOP SCRAPPER RETRACT OUTPUT CUT TIMER
   TOP_SCRP_RET_FLT : BOOL ;	//TOP SCRAPPER RETRACT FAULT
   TOP_SCRP_AUTO_RET_OVR : BOOL ;	//TOP SCRAPPER AUTO RETRACT OVER
   TOP_SCRP_AUTO_RET_DEL : INT  := 3;	//TOP SCRAPPER AUTO RETRACT OVER DELAY
   TOP_SCRP_ATO_RET_DL_T : INT ;	//TOP SCRAPPER AUTO RETRACT OVER DELAY TIMER
   BTM_SCRP_FWD_OP_CUT : BOOL ;	//BOTTOM SCRAPPER FORWARD OUTPUT CUT
   BTM_SCRP_FWD_FLT_TMR : INT ;	//BOTTOM SCRAPPER FORWARD FAULT TIMER
   BTM_SCRP_FWD_FLT_GEN : INT  := 8;	//BOTTOM SCRAPPER FORWARD FAULT GENERATION TIME
   BTM_SCRP_FWD_OP_CT_TM : INT ;	//BOTTOM SCRAPPER FORWARD OUTPUT CUT TIMER
   BTM_SCRP_FWD_FLT : BOOL ;	//BOTTOM SCRAPPER FORWARD FAULT
   BTM_SCRP_AUTO_FWD_OVR : BOOL ;	//BOTTOM SCRAPPER AUTO FORWARD OVER
   BTM_SCRP_AUTO_FWD_DEL : INT  := 3;	//BOTTOM SCRAPPER AUTO FORWARD OVER DELAY
   BTM_SCRP_ATO_FWD_DL_T : INT ;	//BOTTOM SCRAPPER AUTO FORWARD OVER DELAY TIMER
   BTM_SCRP_RET_OP_CUT : BOOL ;	//BOTTOM SCRAPPER RETRACT OUTPUT CUT
   BTM_SCRP_RET_FLT_TMR : INT ;	//BOTTOM SCRAPPER RETRACT FAULT TIMER
   BTM_SCRP_RET_FLT_GEN : INT  := 8;	//BOTTOM SCRAPPER RETRACT FAULT GENERATION TIME
   BTM_SCRP_RET_OP_CT_TM : INT ;	//BOTTOM SCRAPPER RETRACT OUTPUT CUT TIMER
   BTM_SCRP_RET_FLT : BOOL ;	//BOTTOM SCRAPPER RETRACT FAULT
   BTM_SCRP_AUTO_RET_OVR : BOOL ;	//BOTTOM SCRAPPER AUTO RETRACT OVER
   BTM_SCRP_AUTO_RET_DEL : INT  := 3;	//BOTTOM SCRAPPER AUTO RETRACT OVER DELAY
   BTM_SCRP_ATO_RET_DL_T : INT ;	//BOTTOM SCRAPPER AUTO RETRACT OVER DELAY TIMER
   GRV_SCRP_1_FWD_OP_CUT : BOOL ;	//GROOVE SCRAPPER 1 FORWARD OUTPUT CUT
   GRV_SCRP_1_FWD_FLT_TMR : INT ;	//GROOVE SCRAPPER 1 FORWARD FAULT TIMER
   GRV_SCRP_1_FWD_FLT_GEN : INT  := 8;	//GROOVE SCRAPPER 1 FORWARD FAULT GENERATION TIME
   GRV_SCRP_1_FWD_OP_CT_TM : INT ;	//GROOVE SCRAPPER 1 FORWARD OUTPUT CUT TIMER
   GRV_SCRP_1_FWD_FLT : BOOL ;	//GROOVE SCRAPPER 1 FORWARD FAULT
   GRV_SCRP_1_AUTO_FWD_OVR : BOOL ;	//GROOVE SCRAPPER 1 AUTO FORWARD OVER
   GRV_SCRP_1_AUTO_FWD_DEL : INT  := 3;	//GROOVE SCRAPPER 1 AUTO FORWARD OVER DELAY
   GRV_SCRP_1_ATO_FWD_DL_T : INT ;	//GROOVE SCRAPPER 1 AUTO FORWARD OVER DELAY TIMER
   GRV_SCRP_1_RET_OP_CUT : BOOL ;	//GROOVE SCRAPPER 1 RETRACT OUTPUT CUT
   GRV_SCRP_1_RET_FLT_TMR : INT ;	//GROOVE SCRAPPER 1 RETRACT FAULT TIMER
   GRV_SCRP_1_RET_FLT_GEN : INT  := 8;	//GROOVE SCRAPPER 1 RETRACT FAULT GENERATION TIME
   GRV_SCRP_1_RET_OP_CT_TM : INT ;	//GROOVE SCRAPPER 1 RETRACT OUTPUT CUT TIMER
   GRV_SCRP_1_RET_FLT : BOOL ;	//GROOVE SCRAPPER 1 RETRACT FAULT
   GRV_SCRP_1_AUTO_RET_OVR : BOOL ;	//GROOVE SCRAPPER 1 AUTO RETRACT OVER
   GRV_SCRP_1_AUTO_RET_DEL : INT  := 3;	//GROOVE SCRAPPER 1 AUTO RETRACT OVER DELAY
   GRV_SCRP_1_ATO_RET_DL_T : INT ;	//GROOVE SCRAPPER 1 AUTO RETRACT OVER DELAY TIMER
   GRV_SCRP_1_FWD_CMD : BOOL ;	//GROOVE SCRAPPER 1 FORWARD COMMAND
   GRV_SCRP_1_RET_CMD : BOOL ;	//GROOVE SCRAPPER 1 RETRACT COMMAND
   GRV_SCRP_2_FWD_CMD : BOOL ;	//GROOVE SCRAPPER 2 FORWARD COMMAND
   GRV_SCRP_2_RET_CMD : BOOL ;	//GROOVE SCRAPPER 2 RETRACT COMMAND
   GRV_SCRP_1_FWD_LS : BOOL ;	//GROOVE SCRAPPER 1 FORWARD LIMIT SWITCH
   GRV_SCRP_1_RET_LS : BOOL ;	//GROOVE SCRAPPER 1 RETRACT LIMIT SWITCH
   GRV_SCRP_2_FWD_LS : BOOL ;	//GROOVE SCRAPPER 2 FORWARD LIMIT SWITCH
   GRV_SCRP_2_RET_LS : BOOL ;	//GROOVE SCRAPPER 2 RETRACT LIMIT SWITCH
   GRV_SCRP_2_FWD_OP_CUT : BOOL ;	//GROOVE SCRAPPER 2 FORWARD OUTPUT CUT
   GRV_SCRP_2_FWD_FLT_TMR : INT ;	//GROOVE SCRAPPER 2 FORWARD FAULT TIMER
   GRV_SCRP_2_FWD_FLT_GEN : INT  := 8;	//GROOVE SCRAPPER 2 FORWARD FAULT GENERATION TIME
   GRV_SCRP_2_FWD_OP_CT_TM : INT ;	//GROOVE SCRAPPER 2 FORWARD OUTPUT CUT TIMER
   GRV_SCRP_2_FWD_FLT : BOOL ;	//GROOVE SCRAPPER 2 FORWARD FAULT
   GRV_SCRP_2_AUTO_FWD_OVR : BOOL ;	//GROOVE SCRAPPER 2 AUTO FORWARD OVER
   GRV_SCRP_2_AUTO_FWD_DEL : INT  := 3;	//GROOVE SCRAPPER 2 AUTO FORWARD OVER DELAY
   GRV_SCRP_2_ATO_FWD_DL_T : INT ;	//GROOVE SCRAPPER 2 AUTO FORWARD OVER DELAY TIMER
   GRV_SCRP_2_RET_OP_CUT : BOOL ;	//GROOVE SCRAPPER 2 RETRACT OUTPUT CUT
   GRV_SCRP_2_RET_FLT_TMR : INT ;	//GROOVE SCRAPPER 2 RETRACT FAULT TIMER
   GRV_SCRP_2_RET_FLT_GEN : INT  := 8;	//GROOVE SCRAPPER 2 RETRACT FAULT GENERATION TIME
   GRV_SCRP_2_RET_OP_CT_TM : INT ;	//GROOVE SCRAPPER 2 RETRACT OUTPUT CUT TIMER
   GRV_SCRP_2_RET_FLT : BOOL ;	//GROOVE SCRAPPER 2 RETRACT FAULT
   GRV_SCRP_2_AUTO_RET_OVR : BOOL ;	//GROOVE SCRAPPER 2 AUTO RETRACT OVER
   GRV_SCRP_2_AUTO_RET_DEL : INT  := 3;	//GROOVE SCRAPPER 2 AUTO RETRACT OVER DELAY
   GRV_SCRP_2_ATO_RET_DL_T : INT ;	//GROOVE SCRAPPER 2 AUTO RETRACT OVER DELAY TIMER
   CLEAN_OVN_DR_STA : BOOL ;	//CLEAN OVEN DOOR START PUSH BUTTON
   CLEAN_OVN_DR_STP : BOOL ;	//CLEAN OVEN DOOR STOP PUSH BUTTON
   CLEAN_OVN_DR_IND : BOOL ;	//CLEAN OVEN DOOR INDICATION
   CLEAN_OVN_DR_ILK_RDY : BOOL ;	//CLEAN OVEN DOOR INTERLOCK READY FOR START
   CLEAN_OVN_DR_AUTO_STA : BOOL ;	//CLEAN OVEN DOOR AUTO START
   CLEAN_OVN_DR_OPRR_FIN : BOOL ;	//CLEAN OVEN DOOR OPERATIONS FINISHED BIT
   GRV_SRPR_FWD_IND : BOOL ;	//GROOVE SCRAPPER FORWARD INDICATOR
   GRV_SRPR_RET_IND : BOOL ;	//GROOVE SCRAPPER RETRACT INDICATOR
   CLEAN_OVN_DR_HME_POS : BOOL ;	//CLEAN OVEN DOOR HOME POSITION BIT
   BTM_SCRP_AUTO_FWD_SET : BOOL ;	//BOTTOM SCRAPPER AUTO FORWARD SET
   TOP_SCRP_AUTO_FWD_SET : BOOL ;	//TOP SCRAPPER AUTO FORWARD SET
   VER_CLNR_AUTO_CNT : INT ;	//VERTICAL CLEANER CLEANING COUNT
   VER_CLNR_AUTO_CNT_SET : INT  := 2;	//VERTICAL CLEANER CLEANING COUNT SET POINT
   VER_CLNR_AUTO_CNT_OVER : BOOL ;	//VERTICAL CLEANER AUTO COUNT OVER BIT
   GRV_SCRP_FWD_PB : BOOL ;	//GROOVE SCRAPPER FWD PUSH BUTTON CD
   GRV_SCRP_RET_PB : BOOL ;	//GROOVE SCRAPPER RETRACT PUSH BUTTON CD
   BTM_SCRP_AUTO_RET_SET : BOOL ;	//BOTTOM SCRAPPER AUTO RETRACT SET
   TOP_SCRP_AUTO_RET_SET : BOOL ;	//TOP SCRAPPER AUTO RETRACT SET
   CAR_TRA_AUTO_FWD_SET : BOOL ;	//CARRIAGE TRAVEL AUTO FORWARD SET
   CAR_TRA_AUTO_RET_SET : BOOL ;	//CARRIAGE TRAVEL AUTO RETRACT SET
   GRV_SCRP_1_AUTO_FWD_SET : BOOL ;	//GROOVE SCRAPPER 1 AUTO FORWARD SET
   GRV_SCRP_1_AUTO_RET_SET : BOOL ;	//GROOVE SCRAPPER 1 AUTO RETRACT SET
   VER_CLNR_AUTO_UP_SET : BOOL ;	//VERTICAL CLEANER AUTO UP SET
   VER_CLNR_AUTO_DN_SET : BOOL ;	//VERTICAL CLEANER AUTO DOWN SET
   PULSE_17 : BOOL ;	//PULSE 17
   PULSE_18 : BOOL ;	//PULSE 18
   PULSE_19 : BOOL ;	//PULSE 19
   PULSE_20 : BOOL ;	//PULSE 20
   PULSE_21 : BOOL ;	//PULSE 21
   PULSE_22 : BOOL ;	//PULSE 22
   PULSE_23 : BOOL ;	//PULSE 23
   PULSE_24 : BOOL ;	//PULSE 24
   GRV_SCRP_2_AUTO_FWD_SET : BOOL ;	//GROOVE SCRAPPER 2 AUTO FORWARD SET
   GRV_SCRP_2_AUTO_RET_SET : BOOL ;	//GROOVE SCRAPPER 2 AUTO RETRACT SET
   DC_VIBR_AUTO_ON_SET : BOOL ;	//DOOR CLEANER VIBRATOR AUTO ON BIT
   DOOR_CLNR_ATO_STP : BOOL ;	//DOOR CLEANER AUTO STOP BIT
  END_STRUCT ;	
BEGIN
   CAR_TRA_FWD_FLT_GEN := 8;
   CAR_TRA_AUTO_FWD_DEL := 3;
   CAR_TRA_RET_FLT_GEN := 8;
   CAR_TRA_AUTO_RET_DEL := 3;
   VER_CLNR_UP_FLT_GEN := 8;
   VER_CLNR_AUTO_UP_DEL := 3;
   VER_CLNR_DN_FLT_GEN := 8;
   VER_CLNR_AUTO_DN_DEL := 3;
   BTM_BRK_HLDR_DN_FLT_GEN := 8;
   BTM_BRK_HLDR_AUTO_DN_DEL := 3;
   BTM_BRK_HLDR_UP_FLT_GEN := 8;
   BTM_BRK_HLDR_AUTO_UP_DEL := 3;
   TOP_SCRP_FWD_FLT_GEN := 8;
   TOP_SCRP_AUTO_FWD_DEL := 3;
   TOP_SCRP_RET_FLT_GEN := 8;
   TOP_SCRP_AUTO_RET_DEL := 3;
   BTM_SCRP_FWD_FLT_GEN := 8;
   BTM_SCRP_AUTO_FWD_DEL := 3;
   BTM_SCRP_RET_FLT_GEN := 8;
   BTM_SCRP_AUTO_RET_DEL := 3;
   GRV_SCRP_1_FWD_FLT_GEN := 8;
   GRV_SCRP_1_AUTO_FWD_DEL := 3;
   GRV_SCRP_1_RET_FLT_GEN := 8;
   GRV_SCRP_1_AUTO_RET_DEL := 3;
   GRV_SCRP_2_FWD_FLT_GEN := 8;
   GRV_SCRP_2_AUTO_FWD_DEL := 3;
   GRV_SCRP_2_RET_FLT_GEN := 8;
   GRV_SCRP_2_AUTO_RET_DEL := 3;
   VER_CLNR_AUTO_CNT_SET := 3;
END_DATA_BLOCK

DATA_BLOCK "JAMB_CLEANER_DB"	// DB 14
AUTHOR : Kamillas
VERSION : 0.1
  STRUCT
   JC_LOC_SS : BOOL ;	//JAMP CLEANER LOCAL SELECTOR SWITCH
   JC_MAN_SS : BOOL ;	//JAMP CLEANER MANUAL SELECTOR SWITCH
   JC_AUTO_SS : BOOL ;	//JAMP CLEANER AUTO SELECTOR SWITCH
   JC_STOP_PB : BOOL ;	//JAMP CLEANER STOP PUSH BUTTON
   SLEW_FWD_STA_PB : BOOL ;	//SLEW FORWARD START PUSH BUTTON
   SLEW_RET_STA_PB : BOOL ;	//SLEW RETRACT START PUSH BUTTON
   TRA_FWD_STA_PB : BOOL ;	//TRAVEL FORWARD START PUSH BUTTON
   TRA_RET_STA_PB : BOOL ;	//TRAVEL RETRACT START PUSH BUTTON
   VER_CLNR_UP_STA_PB : BOOL ;	//VERTICAL CLEANER UP  START PUSH BUTTON
   VER_CLNR_DN_STA_PB : BOOL ;	//VERTICAL CLEANER DN START PUSH BUTTON
   LCS_90_EMERGENCY_PB : BOOL ;	//LCS-90 EMERGENCY PUSH BUTTON
   SLEW_FWD_STA_PB_LCS : BOOL ;	//SLEW FORWARD START PUSH BUTTON LCS
   SLEW_RET_STA_PB_LCS : BOOL ;	//SLEW RETRACT START PUSH BUTTON LCS
   TRA_FWD_STA_PB_LCS : BOOL ;	//TRAVEL FORWARD START PUSH BUTTON LCS
   TRA_RET_STA_PB_LCS : BOOL ;	//TRAVEL RETRACT START PUSH BUTTON LCS
   VER_CLNR_UP_STA_PB_LCS : BOOL ;	//VERTICAL CLEANER UP  START PUSH BUTTON LCS
   VER_CLNR_DN_STA_PB_LCS : BOOL ;	//VERTICAL CLEANER DN START PUSH BUTTON LCS
   LAMP_TEST_PB_LCS_90 : BOOL ;	//LCS-90 LAMP TEST PUSH BUTTON
   SLEW_SLOW_FWD_LS : BOOL ;	//SLEW SLOW FORWARD LIMIT SWITCH
   SLEW_SLOW_RET_LS : BOOL ;	//SLEW SLOW RETRACT LIMIT SWITCH
   SLEW_NORM_FWD_LS : BOOL ;	//SLEW NORMAL FORWARD LIMIT SWITCH
   SLEW_NORM_RET_LS : BOOL ;	//SLEW NORMAL RETRACT LIMIT SWITCH
   TRA_SLOW_FWD_LS : BOOL ;	//TRAVEL SLOW FORWARD LIMIT  SWITCH
   TRA_SLOW_RET_LS : BOOL ;	//TRAVEL SLOW RETRACT LIMIT  SWITCH
   TRA_NORM_FWD_LS : BOOL ;	//TRAVEL NORMAL FORWARD LIMIT  SWITCH
   TRA_NORM_RET_LS : BOOL ;	//TRAVEL NORMAL RETRACT LIMIT  SWITCH
   VER_CLNR_UP_LS : BOOL ;	//VERTICAL CLEANER UP LIMIIT SWITCH
   VER_CLNR_DN_LS : BOOL ;	//VERTICAL CLEANER DN LIMIIT SWITCH
   SLEW_SLOW_FWD_CMD : BOOL ;	//SLEW SLOW FORWARD COMMAND
   SLEW_SLOW_RET_CMD : BOOL ;	//SLEW SLOW RETRACT COMMAND
   SLEW_NORM_FWD_CMD : BOOL ;	//SLEW NORMAL FORWARD COMMAND
   SLEW_NORM_RET_CMD : BOOL ;	//SLEW NORMAL RETRACT COMMAND
   TRA_SLOW_FWD_CMD : BOOL ;	//TRAVEL SLOW FORWARD COMMAND
   TRA_SLOW_RET_CMD : BOOL ;	//TRAVEL SLOW RETRACT COMMAND
   TRA_NORM_FWD_CMD : BOOL ;	//TRAVEL NORMAL FORWARD COMMAND
   TRA_NORM_RET_CMD : BOOL ;	//TRAVEL NORMAL RETRACT COMMAND
   VER_CLNR_UP_CMD : BOOL ;	//VERTICAL CLEANER UP COMMAND
   VER_CLNR_DN_CMD : BOOL ;	//VERTICAL CLEANER DN COMMAND
   SLEW_FWD_IND : BOOL ;	//SLEW FORWARD INDICATOR
   SLEW_RET_IND : BOOL ;	//SLEW RETRACT INDICATOR
   TRA_FWD_IND : BOOL ;	//TRAVEL FORWARD INDICATOR
   TRA_RET_IND : BOOL ;	//TRAVEL RETRACT INDICATOR
   VER_CLNR_UP_IND : BOOL ;	//VERTICAL CLEANER UP INDICATOR
   VER_CLNR_DN_IND : BOOL ;	//VERTICAL CLEANER DN INDICATOR
   SLEW_FWD_IND_LCS : BOOL ;	//SLEW FORWARD INDICATOR LCS
   SLEW_RET_IND_LCS : BOOL ;	//SLEW RETRACT INDICATOR LCS
   TRA_FWD_IND_LCS : BOOL ;	//TRAVEL FORWARD INDICATOR LCS
   TRA_RET_IND_LCS : BOOL ;	//TRAVEL RETRACT INDICATOR LCS
   VER_CLNR_UP_IND_LCS : BOOL ;	//VERTICAL CLEANER UP INDICATOR LCS
   VER_CLNR_DN_IND_LCS : BOOL ;	//VERTICAL CLEANER DN INDICATOR
   LCS_90_ON_IND : BOOL ;	//LCS-90 ON INDICATOR
   SLEW_SLOW_FWD_OP_CUT : BOOL ;	//SLEW SLOW FORWARD OUTPUT CUT
   SLEW_SLOW_FWD_FLT_TMR : INT ;	//SLEW SLOW FORWARD FAULT TIMER
   SLEW_SLOW_FWD_FLT_GEN : INT  := 8;	//SLEW SLOW FORWARD FAULT GENERATION TIME
   SLEW_SLOW_FWD_OP_CT_TM : INT ;	//SLEW SLOW FORWARD OUTPUT CUT TIMER
   SLEW_SLOW_FWD_FLT : BOOL ;	//SLEW SLOW FORWARD FAULT
   SLEW_SLOW_AUTO_FWD_OVR : BOOL ;	//SLEW SLOW AUTO FORWARD OVER
   SLEW_SLOW_AUTO_FWD_DEL : INT  := 3;	//SLEW SLOW AUTO FORWARD OVER DELAY
   SLEW_SLOW_ATO_FWD_DL_T : INT ;	//SLEW SLOW AUTO FORWARD OVER DELAY TIMER
   SLEW_SLOW_RET_OP_CUT : BOOL ;	//SLEW SLOW RETRACT OUTPUT CUT
   SLEW_SLOW_RET_FLT_TMR : INT ;	//SLEW SLOW RETRACT FAULT TIMER
   SLEW_SLOW_RET_FLT_GEN : INT  := 8;	//SLEW SLOW RETRACT FAULT GENERATION TIME
   SLEW_SLOW_RET_OP_CT_TM : INT ;	//SLEW SLOW RETRACT OUTPUT CUT TIMER
   SLEW_SLOW_RET_FLT : BOOL ;	//SLEW SLOW RETRACT FAULT
   SLEW_SLOW_AUTO_RET_OVR : BOOL ;	//SLEW SLOW AUTO RETRACT OVER
   SLEW_SLOW_AUTO_RET_DEL : INT  := 3;	//SLEW SLOW AUTO RETRACT OVER DELAY
   SLEW_SLOW_ATO_RET_DL_T : INT ;	//SLEW SLOW AUTO RETRACT OVER DELAY TIMER
   SLEW_SLOW_FWD_BIT : BOOL ;	//SLEW SLOW FORWARD START BIT
   SLEW_NORM_FWD_OP_CUT : BOOL ;	//SLEW NORMAL FORWARD OUTPUT CUT
   SLEW_NORM_FWD_FLT_TMR : INT ;	//SLEW NORMAL FORWARD FAULT TIMER
   SLEW_NORM_FWD_FLT_GEN : INT  := 8;	//SLEW NORMAL FORWARD FAULT GENERATION TIME
   SLEW_NORM_FWD_OP_CT_TM : INT ;	//SLEW NORMAL FORWARD OUTPUT CUT TIMER
   SLEW_NORM_FWD_FLT : BOOL ;	//SLEW NORMAL FORWARD FAULT
   SLEW_NORM_AUTO_FWD_OVR : BOOL ;	//SLEW NORMAL AUTO FORWARD OVER
   SLEW_NORM_AUTO_FWD_DEL : INT  := 3;	//SLEW NORMAL AUTO FORWARD OVER DELAY
   SLEW_NORM_ATO_FWD_DL_T : INT ;	//SLEW NORMAL AUTO FORWARD OVER DELAY TIMER
   SLEW_NORM_RET_OP_CUT : BOOL ;	//SLEW NORMAL RETRACT OUTPUT CUT
   SLEW_NORM_RET_FLT_TMR : INT ;	//SLEW NORMAL RETRACT FAULT TIMER
   SLEW_NORM_RET_FLT_GEN : INT  := 8;	//SLEW NORMAL RETRACT FAULT GENERATION TIME
   SLEW_NORM_RET_OP_CT_TM : INT ;	//SLEW NORMAL RETRACT OUTPUT CUT TIMER
   SLEW_NORM_RET_FLT : BOOL ;	//SLEW NORMAL RETRACT FAULT
   SLEW_NORM_AUTO_RET_OVR : BOOL ;	//SLEW NORMAL AUTO RETRACT OVER
   SLEW_NORM_AUTO_RET_DEL : INT  := 3;	//SLEW NORMAL AUTO RETRACT OVER DELAY
   SLEW_NORM_ATO_RET_DL_T : INT ;	//SLEW NORMAL AUTO RETRACT OVER DELAY TIMER
   PULSE_1 : BOOL ;	//PULSE 1
   PULSE_2 : BOOL ;	//PULSE 2
   PULSE_3 : BOOL ;	//PULSE 3
   PULSE_4 : BOOL ;	//PULSE 4
   PULSE_5 : BOOL ;	//PULSE 5
   PULSE_6 : BOOL ;	//PULSE 6
   PULSE_7 : BOOL ;	//PULSE 7
   PULSE_8 : BOOL ;	//PULSE 8
   PULSE_9 : BOOL ;	//PULSE 9
   PULSE_10 : BOOL ;	//PULSE 10
   PULSE_11 : BOOL ;	//PULSE 11
   PULSE_12 : BOOL ;	//PULSE 12
   PULSE_13 : BOOL ;	//PULSE 13
   PULSE_14 : BOOL ;	//PULSE 14
   PULSE_15 : BOOL ;	//PULSE 15
   PULSE_16 : BOOL ;	//PULSE 16
   TRA_SLOW_FWD_OP_CUT : BOOL ;	//TRAVEL SLOW FORWARD OUTPUT CUT
   TRA_SLOW_FWD_FLT_TMR : INT ;	//TRAVEL SLOW FORWARD FAULT TIMER
   TRA_SLOW_FWD_FLT_GEN : INT  := 8;	//TRAVEL SLOW FORWARD FAULT GENERATION TIME
   TRA_SLOW_FWD_OP_CT_TM : INT ;	//TRAVEL SLOW FORWARD OUTPUT CUT TIMER
   TRA_SLOW_FWD_FLT : BOOL ;	//TRAVEL SLOW FORWARD FAULT
   TRA_SLOW_AUTO_FWD_OVR : BOOL ;	//TRAVEL SLOW AUTO FORWARD OVER
   TRA_SLOW_AUTO_FWD_DEL : INT  := 3;	//TRAVEL SLOW AUTO FORWARD OVER DELAY
   TRA_SLOW_ATO_FWD_DL_T : INT ;	//TRAVEL SLOW AUTO FORWARD OVER DELAY TIMER
   TRA_SLOW_RET_OP_CUT : BOOL ;	//TRAVEL SLOW RETRACT OUTPUT CUT
   TRA_SLOW_RET_FLT_TMR : INT ;	//TRAVEL SLOW RETRACT FAULT TIMER
   TRA_SLOW_RET_FLT_GEN : INT  := 8;	//TRAVEL SLOW RETRACT FAULT GENERATION TIME
   TRA_SLOW_RET_OP_CT_TM : INT ;	//TRAVEL SLOW RETRACT OUTPUT CUT TIMER
   TRA_SLOW_RET_FLT : BOOL ;	//TRAVEL SLOW RETRACT FAULT
   TRA_SLOW_AUTO_RET_OVR : BOOL ;	//TRAVEL SLOW AUTO RETRACT OVER
   TRA_SLOW_AUTO_RET_DEL : INT  := 3;	//TRAVEL SLOW AUTO RETRACT OVER DELAY
   TRA_SLOW_ATO_RET_DL_T : INT ;	//TRAVEL SLOW AUTO RETRACT OVER DELAY TIMER
   TRA_SLOW_FWD_BIT : BOOL ;	//TRAVEL SLOW FORWARD START BIT
   TRA_NORM_FWD_OP_CUT : BOOL ;	//TRAVEL NORMAL FORWARD OUTPUT CUT
   TRA_NORM_FWD_FLT_TMR : INT ;	//TRAVEL NORMAL FORWARD FAULT TIMER
   TRA_NORM_FWD_FLT_GEN : INT  := 8;	//TRAVEL NORMAL FORWARD FAULT GENERATION TIME
   TRA_NORM_FWD_OP_CT_TM : INT ;	//TRAVEL NORMAL FORWARD OUTPUT CUT TIMER
   TRA_NORM_FWD_FLT : BOOL ;	//TRAVEL NORMAL FORWARD FAULT
   TRA_NORM_AUTO_FWD_OVR : BOOL ;	//TRAVEL NORMAL AUTO FORWARD OVER
   TRA_NORM_AUTO_FWD_DEL : INT  := 3;	//TRAVEL NORMAL AUTO FORWARD OVER DELAY
   TRA_NORM_ATO_FWD_DL_T : INT ;	//TRAVEL NORMAL AUTO FORWARD OVER DELAY TIMER
   TRA_NORM_RET_OP_CUT : BOOL ;	//TRAVEL NORMAL RETRACT OUTPUT CUT
   TRA_NORM_RET_FLT_TMR : INT ;	//TRAVEL NORMAL RETRACT FAULT TIMER
   TRA_NORM_RET_FLT_GEN : INT  := 8;	//TRAVEL NORMAL RETRACT FAULT GENERATION TIME
   TRA_NORM_RET_OP_CT_TM : INT ;	//TRAVEL NORMAL RETRACT OUTPUT CUT TIMER
   TRA_NORM_RET_FLT : BOOL ;	//TRAVEL NORMAL RETRACT FAULT
   TRA_NORM_AUTO_RET_OVR : BOOL ;	//TRAVEL NORMAL AUTO RETRACT OVER
   TRA_NORM_AUTO_RET_DEL : INT  := 3;	//TRAVEL NORMAL AUTO RETRACT OVER DELAY
   TRA_NORM_ATO_RET_DL_T : INT ;	//TRAVEL NORMAL AUTO RETRACT OVER DELAY TIMER
   VER_CLNR_FWD_OP_CUT : BOOL ;	//VERTICAL CLEANER FORWARD OUTPUT CUT
   VER_CLNR_FWD_FLT_TMR : INT ;	//VERTICAL CLEANER FORWARD FAULT TIMER
   VER_CLNR_FWD_FLT_GEN : INT  := 8;	//VERTICAL CLEANER FORWARD FAULT GENERATION TIME
   VER_CLNR_FWD_OP_CT_TM : INT ;	//VERTICAL CLEANER FORWARD OUTPUT CUT TIMER
   VER_CLNR_FWD_FLT : BOOL ;	//VERTICAL CLEANER FORWARD FAULT
   VER_CLNR_AUTO_FWD_OVR : BOOL ;	//VERTICAL CLEANER AUTO FORWARD OVER
   VER_CLNR_AUTO_FWD_DEL : INT  := 3;	//VERTICAL CLEANER AUTO FORWARD OVER DELAY
   VER_CLNR_ATO_FWD_DL_T : INT ;	//VERTICAL CLEANER AUTO FORWARD OVER DELAY TIMER
   VER_CLNR_RET_OP_CUT : BOOL ;	//VERTICAL CLEANER RETRACT OUTPUT CUT
   VER_CLNR_RET_FLT_TMR : INT ;	//VERTICAL CLEANER RETRACT FAULT TIMER
   VER_CLNR_RET_FLT_GEN : INT  := 8;	//VERTICAL CLEANER RETRACT FAULT GENERATION TIME
   VER_CLNR_RET_OP_CT_TM : INT ;	//VERTICAL CLEANER RETRACT OUTPUT CUT TIMER
   VER_CLNR_RET_FLT : BOOL ;	//VERTICAL CLEANER RETRACT FAULT
   VER_CLNR_AUTO_RET_OVR : BOOL ;	//VERTICAL CLEANER AUTO RETRACT OVER
   VER_CLNR_AUTO_RET_DEL : INT  := 3;	//VERTICAL CLEANER AUTO RETRACT OVER DELAY
   VER_CLNR_ATO_RET_DL_T : INT ;	//VERTICAL CLEANER AUTO RETRACT OVER DELAY TIMER
   TRA_SLOW_FWD_IND_LCS : BOOL ;	//TRAVEL SLOW FORWARD INDICATOR LCS
   TRA_SLOW_RET_IND_LCS : BOOL ;	//TRAVEL SLOW RETRACT INDICATOR LCS
   TRA_SLOW_FWD_IND : BOOL ;	//TRAVEL SLOW FORWARD INDICATOR
   TRA_SLOW_RET_IND : BOOL ;	//TRAVEL SLOW RETRACT INDICATOR
   JAMB_CLNR_AUTO_STA_PB : BOOL ;	//JAMB CLEANER AUTO START PUSH BUTTON
   JAMB_CLNR_AUTO_STP_PB : BOOL ;	//JAMB CLEANER AUTO STOP PUSH BUTTON
   JC_SLEW_AUTO_FWD_SET : BOOL ;	//JAMB CLEANER SLEW AUTO FORWARD SET
   JC_SLEW_AUTO_RET_SET : BOOL ;	//JAMB CLEANER SLEW AUTO RETRACT SET
   JC_TRA_AUTO_FWD_SET : BOOL ;	//JAMB CLEANER TRAVEL AUTO FORWARD SET
   JC_TRA_AUTO_RET_SET : BOOL ;	//JAMB CLEANER TRAVEL AUTO RETRACT SET
   VER_CLNT_AUTO_CNT_OVER : BOOL ;	//JAMB CLEANER VERTICAL CLEANER AUTO COUNT OVER
   VER_CLNR_AUTO_COUNT : INT ;	//JAMB CLEANER AUTO COUNT
   VER_CLNR_AUTO_COUNT_SET : INT  := 2;	//JAMB CLEANER AUTO COUNT SET POINT
   JAMB_CLNR_ILK : BOOL ;	//JAMB CLEANER INTERLOCK BIT
   JAMB_CLNR_IND : BOOL ;	//JAMB CLEANER INDICATOR
   JAMB_CLNR_AUTO_STA : BOOL ;	//JAMB CLEANER AUTO START
   VER_CLNR_AUTO_FWD_SET : BOOL ;	//VERTICAL CLEANER AUTO FORWARD SET
   VER_CLNR_AUTO_RET_SET : BOOL ;	//VERTICAL CLEANER AUTO RETRACT SET
   JAMB_CLNR_HME_POS : BOOL ;	//JAMB CLEANER HOME POSITION BIT
   JAMB_CLNR_OVN_OPER_FIN : BOOL ;	//JAMB CLEANER CLEAN OVEN OPERATIONS FISISHED
   JAMB_CLNR_AUTO_MID_STOP : BOOL ;	//JAMB CLEANER AUTO OPERATIONS STOPPER WHILE IN AUTO OPERATION
  END_STRUCT ;	
BEGIN
   SLEW_SLOW_FWD_FLT_GEN := 8;
   SLEW_SLOW_AUTO_FWD_DEL := 3;
   SLEW_SLOW_RET_FLT_GEN := 8;
   SLEW_SLOW_AUTO_RET_DEL := 3;
   SLEW_NORM_FWD_FLT_GEN := 8;
   SLEW_NORM_AUTO_FWD_DEL := 3;
   SLEW_NORM_RET_FLT_GEN := 8;
   SLEW_NORM_AUTO_RET_DEL := 3;
   TRA_SLOW_FWD_FLT_GEN := 8;
   TRA_SLOW_AUTO_FWD_DEL := 3;
   TRA_SLOW_RET_FLT_GEN := 8;
   TRA_SLOW_AUTO_RET_DEL := 3;
   TRA_NORM_FWD_FLT_GEN := 8;
   TRA_NORM_AUTO_FWD_DEL := 3;
   TRA_NORM_RET_FLT_GEN := 8;
   TRA_NORM_AUTO_RET_DEL := 3;
   VER_CLNR_FWD_FLT_GEN := 8;
   VER_CLNR_AUTO_FWD_DEL := 3;
   VER_CLNR_RET_FLT_GEN := 8;
   VER_CLNR_AUTO_RET_DEL := 3;
   VER_CLNR_AUTO_COUNT_SET := 2;
END_DATA_BLOCK

DATA_BLOCK "COUNTER_THRUST_WEDGE_DB"	// DB 15
AUTHOR : Kamillas
VERSION : 0.1
  STRUCT
   CNT_TH_WED_LOC_SS : BOOL ;	//COUNTER THRUST WEDGE LOCAL SELECTOR SWITCH
   CNT_TH_WED_MAN_SS : BOOL ;	//COUNTER THRUST WEDGE MAUAL SELECTOR SWITCH
   CNT_TH_WED_AUTO_SS : BOOL ;	//COUNTER THRUST WEDGE AUTO SELECTOR SWITCH
   CNT_TH_WED_STOP_PB : BOOL ;	//COUNTER THRUST WEDGE STOP PUSH BUTTON
   CNT_TH_WED_UP_STA_PB : BOOL ;	//COUNTER THRUST WEDGE UP START PUSH BUTTON
   CNT_TH_WED_DN_STA_PB : BOOL ;	//COUNTER THRUST WEDGE DN START PUSH BUTTON
   CNT_TH_WED_DN_STA_PB_LCS : BOOL ;	//COUNTER THRUST WEDGE DN START PUSH BUTTON LCS
   CNT_TH_WED_UP_STA_PB_LCS : BOOL ;	//COUNTER THRUST WEDGE UP START PUSH BUTTON LCS
   EMEG_STOP_PB_LCS_72 : BOOL ;	//EMERGENCY STOP PUSH BUTTON LCS-72
   CNT_TH_WED1_DN_LS : BOOL ;	//COUNTER THRUST WEDGE-1 DN  LIMIT SWITCH
   CNT_TH_WED1_UP_LS : BOOL ;	//COUNTER THRUST WEDGE-1 UP  LIMIT SWITCH
   CNT_TH_WED2_DN_LS : BOOL ;	//COUNTER THRUST WEDGE-2 DN LIMIT SWITCH
   CNT_TH_WED2_UP_LS : BOOL ;	//COUNTER THRUST WEDGE-2 UP LIMIT SWITCH
   CNT_TH_WED_UP_CMD : BOOL ;	//COUNTER THRUST WEDGE UP COMMAND
   CNT_TH_WED_DN_CMD : BOOL ;	//COUNTER THRUST WEDGE DN COMMAND
   CNT_TH_WED_UP_IND : BOOL ;	//COUNTER THRUST WEDGE UP INDICATOR
   CNT_TH_WED_DN_IND : BOOL ;	//COUNTER THRUST WEDGE DN INDICATOR
   CNT_TH_WED_UP_IND_LCS : BOOL ;	//COUNTER THRUST WEDGE UP INDICATOR LCS
   CNT_TH_WED_DN_IND_LCS : BOOL ;	//COUNTER THRUST WEDGE DN INDICATOR LCS
   CNT_TH_WED_LOC_IND_LCS : BOOL ;	//COUNTER THRUST WEDGE LOCAL INDICATOR LCS
   CNT_TH_WED_UP_OP_CUT : BOOL ;	//COUNTER THRUST WEDGE UP OUTPUT CUT
   CNT_TH_WED_UP_FLT_TMR : INT ;	//COUNTER THRUST WEDGE UP FAULT TIMER
   CNT_TH_WED_UP_FLT_GEN : INT  := 8;	//COUNTER THRUST WEDGE UP FAULT GENERATION TIME
   CNT_TH_WED_UP_OP_CT_TM : INT ;	//COUNTER THRUST WEDGE UP OUTPUT CUT TIMER
   CNT_TH_WED_UP_FLT : BOOL ;	//COUNTER THRUST WEDGE UP FAULT
   CNT_TH_WED_AUTO_UP_OVR : BOOL ;	//COUNTER THRUST WEDGE AUTO UP OVER
   CNT_TH_WED_AUTO_UP_DEL : INT  := 3;	//COUNTER THRUST WEDGE AUTO UP OVER DELAY
   CNT_TH_WED_ATO_UP_DL_T : INT ;	//COUNTER THRUST WEDGE AUTO UP OVER DELAY TIMER
   CNT_TH_WED_DN_OP_CUT : BOOL ;	//COUNTER THRUST WEDGE DOWN OUTPUT CUT
   CNT_TH_WED_DN_FLT_TMR : INT ;	//COUNTER THRUST WEDGE DOWN FAULT TIMER
   CNT_TH_WED_DN_FLT_GEN : INT  := 8;	//COUNTER THRUST WEDGE DOWN FAULT GENERATION TIME
   CNT_TH_WED_DN_OP_CT_TM : INT ;	//COUNTER THRUST WEDGE DOWN OUTPUT CUT TIMER
   CNT_TH_WED_DN_FLT : BOOL ;	//COUNTER THRUST WEDGE DOWN FAULT
   CNT_TH_WED_AUTO_DN_OVR : BOOL ;	//COUNTER THRUST WEDGE AUTO DOWN OVER
   CNT_TH_WED_AUTO_DN_DEL : INT  := 3;	//COUNTER THRUST WEDGE AUTO DOWN OVER DELAY
   CNT_TH_WED_ATO_DN_DL_T : INT ;	//COUNTER THRUST WEDGE AUTO DOWN OVER DELAY TIMER
   PULSE_1 : BOOL ;	//PULSE 1
   PULSE_2 : BOOL ;	//PULSE 2
   PULSE_3 : BOOL ;	//PULSE 3
   PULSE_4 : BOOL ;	//PULSE 4
   PULSE_5 : BOOL ;	//PULSE 5
   PULSE_6 : BOOL ;	//PULSE 6
   PULSE_7 : BOOL ;	//PULSE 7
   PULSE_8 : BOOL ;	//PULSE 8
   CNT_TH_WED_SYS_RDY : BOOL ;	//COUNTER THRUST WEDGE SYSTEM READY BIT
   CNT_TH_WED_PREP_AUTO_STA : BOOL ;	//COUNTER THRUST WEDGE PREPARE AUTO START BIT
   PREP_DOOR_FUNC_STA : BOOL ;	//PREPARE DOOR FUNCTION START PUSH BUTTON
   PREP_DOOR_FUNC_STP : BOOL ;	//PREPARE DOOR FUNCTION STOP PUSH BUTTON
   FIN_DOOR_FUNC_STA : BOOL ;	//FINISH DOOR FUNCTION START PUSH BUTTON
   CNT_TH_WED_FIN_AUTO_STA : BOOL ;	//COUNTER THRUST WEDGE FIN AUTO START BIT
   PREP_DOOR_FUNC_IND : BOOL ;	//COUNTER THRUST WEDGE PREPARE DOOR FUNCTION INDICATION
   FIN_DOOR_FUNC_IND : BOOL ;	//COUNTER THRUST WEDGE FINISH DOOR FUNCTION INDICATION
  END_STRUCT ;	
BEGIN
   CNT_TH_WED_UP_FLT_GEN := 8;
   CNT_TH_WED_AUTO_UP_DEL := 3;
   CNT_TH_WED_DN_FLT_GEN := 8;
   CNT_TH_WED_AUTO_DN_DEL := 3;
END_DATA_BLOCK

DATA_BLOCK "COAL_SPILLAGE_SYSTEM_DB"	// DB 16
AUTHOR : Kamillas
VERSION : 0.1
  STRUCT
   CL_SPI_CHT_DN_STA : BOOL ;	//COAL SPILLAGE CHUTE DOWN START PUSH BUTTON
   CL_SPI_CHT_UP_STA : BOOL ;	//COAL SPILLAGE CHUTE UP START PUSH BUTTON
   CL_SPI_CHT_DN_STA_LCS : BOOL ;	//COAL SPILLAGE CHUTE DOWN START PUSH BUTTON LCS
   CL_SPI_CHT_UP_STA_LCS : BOOL ;	//COAL SPILLAGE CHUTE UP START PUSH BUTTON LCS
   CL_SPI_HOP_GT_OP_STA_LCS : BOOL ;	//COAL SPILLAGE HOPPER GATE OPEN START PUSH BUTTON LCS
   CL_SPI_HOP_GT_CL_STA_LCS : BOOL ;	//COAL SPILLAGE HOPPER GATE CLOSE START PUSH BUTTON LCS
   CL_SPI_CHT_DN_LS : BOOL ;	//COAL SPILLAGE CHUTE DOWN LIMIT SWITCH
   CL_SPI_CHT_UP_LS : BOOL ;	//COAL SPILLAGE CHUTE UP LIMIT SWITCH
   CL_SPI_HPR_GT_O_LS : BOOL ;	//COAL SPILLAGE HOPPER GATE OPEN LIMIT SWITCH
   CL_SPI_HPR_GT_C_LS : BOOL ;	//COAL SPILLAGE HOPPER GATE CLOSE LIMIT SWITCH
   CK_SPI_SH_SL_FW_STA_PB : BOOL ;	//COKE SPILLAGE SHOVEL SLEW FORWARD START PUSH BUTTON
   CK_SPI_SH_SL_RT_STA_PB : BOOL ;	//COKE SPILLAGE SHOVEL SLEW RETRACT START PUSH BUTTON
   CK_SPI_SH_SL_FW_STA_LCS : BOOL ;	//COKE SPILLAGE SHOVEL SLEW FORWARD START PUSH BUTTON LCS
   CK_SPI_SH_SL_RT_STA_LCS : BOOL ;	//COKE SPILLAGE SHOVEL SLEW RETRACT START PUSH BUTTON LCS
   CK_SPI_SH_SL_FW_LS : BOOL ;	//COKE SPILLAGE SHOVEL SLEW FORWARD LIMIT SWITCH
   CK_SPI_SH_SL_RT_LS : BOOL ;	//COKE SPILLAGE SHOVEL SLEW RETRACT LIMIT SWITCH
   DR_CL_SH_SL_FWD_STA : BOOL ;	//DOOR CLEANER SPILLAGE SHOWEL SLEW FORWARD PUSH BUTTON START
   DR_CL_SH_SL_RET_STA : BOOL ;	//DOOR CLEANER SPILLAGE SHOWEL SLEW RETRACT PUSH BUTTON START
   DR_CL_SH_SL_FWD_LCS : BOOL ;	//DOOR CLEANER SPILLAGE SHOWEL SLEW FORWARD START PUSH BUTTON LCS
   DR_CL_SH_SL_RET_LCS : BOOL ;	//DOOR CLEANER SPILLAGE SHOWEL SLEW RETRACT START PUSH BUTTON LCS
   DR_CL_SP_HPR_FWD_STA_LCS : BOOL ;	//DOOR CLEANER SPILLAGE HOPPER FORWARD START PUSH BUTTON LCS
   DR_CL_SP_HPR_RET_STA_LCS : BOOL ;	//DOOR CLEANER SPILLAGE HOPPER RETRACT START PUSH BUTTON LCS
   DR_CL_SH_SL_FWD_FB : BOOL ;	//DOOR CLEANER SPILLAGE SHOWEL SLEW FORWARD FEED BACK
   DR_CL_SH_SL_RET_FB : BOOL ;	//DOOR CLEANER SPILLAGE SHOWEL SLEW RETRACT FEED BACK
   DR_CL_SP_HPR_FWD_FB : BOOL ;	//DOOR CLEANER SPILLAGE HOPPER FORWARD FEED BACK
   DR_CL_SP_HPR_RET_FB : BOOL ;	//DOOR CLEANER SPILLAGE HOPPER RETRACT FEED BACK
   CL_SPI_CHT_UP_CMD : BOOL ;	//COAL SPILLAGE CHUTE UP COMMAND
   CL_SPI_CHT_DN_CMD : BOOL ;	//COAL SPILLAGE CHUTE DOWN COMMAND
   CL_SPI_HPR_GT_O_CMD : BOOL ;	//COAL SPILLAGE HOPPER GATE OPEN COMMAND
   CL_SPI_HPR_GT_C_CMD : BOOL ;	//COAL SPILLAGE HOPPER GATE CLOSE COMMAND
   CL_SPI_CHT_UP_IND : BOOL ;	//COAL SPILLAGE CHUTE UP INDICATOR
   CL_SPI_CHT_DN_IND : BOOL ;	//COAL SPILLAGE CHUTE DN INDICATOR
   CL_SPI_CHT_UP_IND_LCS : BOOL ;	//COAL SPILLAGE CHUTE UP INDICATOR LCS
   CL_SPI_CHT_DN_IND_LCS : BOOL ;	//COAL SPILLAGE CHUTE DN INDICATOR LCS
   CL_SPI_HPR_GT_O_IND_LCS : BOOL ;	//COAL SPILLAGE HOPPER GATE OPEN INDICATOR LCS
   CL_SPI_HPR_GT_C_IND_LCS : BOOL ;	//COAL SPILLAGE HOPPER GATE CLOSE INDICATOR LCS
   CK_SPI_SH_SL_FW_CMD : BOOL ;	//COKE SPILLAGE SHOVEL SLEW FORWARD COMMAND
   CK_SPI_SH_SL_RT_CMD : BOOL ;	//COKE SPILLAGE SHOVEL SLEW RETRACT COMMAND
   CK_SPI_SH_SL_FW_IND : BOOL ;	//COKE SPILLAGE SHOVEL SLEW FORWARD INDICATOR
   CK_SPI_SH_SL_RT_IND : BOOL ;	//COKE SPILLAGE SHOVEL SLEW RETRACT INDICATOR
   CK_SPI_SH_SL_FW_IND_LCS : BOOL ;	//COKE SPILLAGE SHOVEL SLEW FORWARD INDICATOR LCS
   CK_SPI_SH_SL_RT_IND_LCS : BOOL ;	//COKE SPILLAGE SHOVEL SLEW RETRACT INDICATOR LCS
   DR_CL_SH_SL_FWD_CMD : BOOL ;	//DOOR CLEANER SPILLAGE SHOWEL SLEW FORWARD COMMAND
   DR_CL_SH_SL_RET_CMD : BOOL ;	//DOOR CLEANER SPILLAGE SHOWEL SLEW RETRACT COMMAND
   DR_CL_SP_HO_FWD_COM : BOOL ;	//DOOR CLEANER SPILLAGE HOPPER FORWARD COMMAND
   DR_CL_SP_HO_RET_COM : BOOL ;	//DOOR CLEANER SPILLAGE HOPPER RETRACT COMMAND
   DR_CL_SH_SL_FWD_IND : BOOL ;	//DOOR CLEANER SPILLAGE SHOWEL SLEW FORWARD INDICATOR
   DR_CL_SH_SL_RET_IND : BOOL ;	//DOOR CLEANER SPILLAGE SHOWEL SLEW RETRACT INDICATOR
   DR_CL_SH_SL_FWD_IND_LCS : BOOL ;	//DOOR CLEANER SPILLAGE SHOWEL SLEW FORWARD INDICATOR LCS
   DR_CL_SH_SL_RET_IND_LCS : BOOL ;	//DOOR CLEANER SPILLAGE SHOWEL SLEW RETRACT INDICATOR LCS
   DR_CL_SP_HPR_FWD_IND : BOOL ;	//DOOR CLEANER SPILLAGE HOPPER FORWARD INDICATOR
   DR_CL_SP_HPR_RET_IND : BOOL ;	//DOOR CLEANER SPILLAGE HOPPER RETRACT INDICATOR
   CL_SPI_CHT_DN_OP_CUT : BOOL ;	//COAL SPILLAGE CHUTE DOWN OUTPUT CUT
   CL_SPI_CHT_DN_FLT_TMR : INT ;	//COAL SPILLAGE CHUTE DOWN FAULT TIMER
   CL_SPI_CHT_DN_FLT_GEN : INT  := 8;	//COAL SPILLAGE CHUTE DOWN FAULT GENERATION TIME
   CL_SPI_CHT_DN_OP_CT_TM : INT ;	//COAL SPILLAGE CHUTE DOWN OUTPUT CUT TIMER
   CL_SPI_CHT_DN_FLT : BOOL ;	//COAL SPILLAGE CHUTE DOWN FORWARD FAULT
   CL_SPI_CHT_AUTO_DN_OVR : BOOL ;	//COAL SPILLAGE CHUTE AUTO DOWN OVER
   CL_SPI_CHT_AUTO_DN_DEL : INT  := 3;	//COAL SPILLAGE CHUTE AUTO DOWN OVER DELAY
   CL_SPI_CHT_ATO_DN_DL_T : INT ;	//COAL SPILLAGE CHUTE AUTO DOWN OVER DELAY TIMER
   PUSLE_1 : BOOL ;	//PULSE 1
   PUSLE_2 : BOOL ;	//PULSE 2
   PUSLE_3 : BOOL ;	//PULSE 3
   PUSLE_4 : BOOL ;	//PULSE 4
   PUSLE_5 : BOOL ;	//PULSE 5
   PUSLE_6 : BOOL ;	//PULSE 6
   PUSLE_7 : BOOL ;	//PULSE 7
   PUSLE_8 : BOOL ;	//PULSE 8
   PUSLE_9 : BOOL ;	//PULSE 9
   PUSLE_10 : BOOL ;	//PULSE 10
   PUSLE_11 : BOOL ;	//PULSE 11
   PUSLE_12 : BOOL ;	//PULSE 12
   PUSLE_13 : BOOL ;	//PULSE 13
   PUSLE_14 : BOOL ;	//PULSE 14
   PUSLE_15 : BOOL ;	//PULSE 15
   PUSLE_16 : BOOL ;	//PULSE 16
   CL_SPI_CHT_UP_OP_CUT : BOOL ;	//COAL SPILLAGE CHUTE UP OUTPUT CUT
   CL_SPI_CHT_UP_FLT_TMR : INT ;	//COAL SPILLAGE CHUTE UP FAULT TIMER
   CL_SPI_CHT_UP_FLT_GEN : INT  := 8;	//COAL SPILLAGE CHUTE UP FAULT GENERATION TIME
   CL_SPI_CHT_UP_OP_CT_TM : INT ;	//COAL SPILLAGE CHUTE UP OUTPUT CUT TIMER
   CL_SPI_CHT_UP_FLT : BOOL ;	//COAL SPILLAGE CHUTE UP FORWARD FAULT
   CL_SPI_CHT_AUTO_UP_OVR : BOOL ;	//COAL SPILLAGE CHUTE AUTO UP OVER
   CL_SPI_CHT_AUTO_UP_DEL : INT  := 3;	//COAL SPILLAGE CHUTE AUTO UP OVER DELAY
   CL_SPI_CHT_ATO_UP_DL_T : INT ;	//COAL SPILLAGE CHUTE AUTO UP OVER DELAY TIMER
   CL_SPI_HPR_GT_O_OP_CUT : BOOL ;	//COAL SPILLAGE HOPPER GATE OPEN OUTPUT CUT
   CL_SPI_HPR_GT_O_FLT_TMR : INT ;	//COAL SPILLAGE HOPPER GATE OPEN FAULT TIMER
   CL_SPI_HPR_GT_O_FLT_GEN : INT  := 8;	//COAL SPILLAGE HOPPER GATE OPEN FAULT GENERATION TIME
   CL_SPI_HPR_GT_O_OP_CT_TM : INT ;	//COAL SPILLAGE HOPPER GATE OPEN OUTPUT CUT TIMER
   CL_SPI_HPR_GT_O_FLT : BOOL ;	//COAL SPILLAGE HOPPER GATE OPEN FORWARD FAULT
   CL_SPI_HPR_GT_AUTO_O_OVR : BOOL ;	//COAL SPILLAGE HOPPER GATE AUTO OPEN OVER
   CL_SPI_HPR_GT_AUTO_O_DEL : INT  := 3;	//COAL SPILLAGE HOPPER GATE AUTO OPEN OVER DELAY
   CL_SPI_HPR_GT_ATO_O_DL_T : INT ;	//COAL SPILLAGE HOPPER GATE AUTO OPEN OVER DELAY TIMER
   CL_SPI_HPR_GT_C_OP_CUT : BOOL ;	//COAL SPILLAGE HOPPER GATE CLOSE OUTPUT CUT
   CL_SPI_HPR_GT_C_FLT_TMR : INT ;	//COAL SPILLAGE HOPPER GATE CLOSE FAULT TIMER
   CL_SPI_HPR_GT_C_FLT_GEN : INT  := 8;	//COAL SPILLAGE HOPPER GATE CLOSE FAULT GENERATION TIME
   CL_SPI_HPR_GT_C_OP_CT_TM : INT ;	//COAL SPILLAGE HOPPER GATE CLOSE OUTPUT CUT TIMER
   CL_SPI_HPR_GT_C_FLT : BOOL ;	//COAL SPILLAGE HOPPER GATE CLOSE FORWARD FAULT
   CL_SPI_HPR_GT_AUTO_C_OVR : BOOL ;	//COAL SPILLAGE HOPPER GATE AUTO CLOSE OVER
   CL_SPI_HPR_GT_AUTO_C_DEL : INT  := 3;	//COAL SPILLAGE HOPPER GATE AUTO CLOSE OVER DELAY
   CL_SPI_HPR_GT_ATO_C_DL_T : INT ;	//COAL SPILLAGE HOPPER GATE AUTO CLOSE OVER DELAY TIMER
   CK_SPI_SH_SL_FW_OP_CUT : BOOL ;	//COKE SPILLAGE SHOVEL SLEW FORWARD OUTPUT CUT
   CK_SPI_SH_SL_FW_FLT_TMR : INT ;	//COKE SPILLAGE SHOVEL SLEW FORWARD FAULT TIMER
   CK_SPI_SH_SL_FW_FLT_GEN : INT  := 8;	//COKE SPILLAGE SHOVEL SLEW FORWARD FAULT GENERATION TIME
   CK_SPI_SH_SL_FW_OP_CT_T : INT ;	//COKE SPILLAGE SHOVEL SLEW FORWARD OUTPUT CUT TIMER
   CK_SPI_SH_SL_FW_FLT : BOOL ;	//COKE SPILLAGE SHOVEL SLEW FORWARD FAULT
   CK_SPI_SH_SL_AUTO_FW_OVR : BOOL ;	//COKE SPILLAGE SHOVEL SLEW AUTO FORWARD OVER
   CK_SPI_SH_SL_AUTO_FW_DEL : INT  := 3;	//COKE SPILLAGE SHOVEL SLEW AUTO FORWARD OVER DELAY
   CK_SPI_SH_SL_ATO_FW_DL_T : INT ;	//COKE SPILLAGE SHOVEL SLEW AUTO FORWARD OVER DELAY TIMER
   CK_SPI_SH_SL_RT_OP_CUT : BOOL ;	//COKE SPILLAGE SHOVEL SLEW RETRACT OUTPUT CUT
   CK_SPI_SH_SL_RT_FLT_TMR : INT ;	//COKE SPILLAGE SHOVEL SLEW RETRACT FAULT TIMER
   CK_SPI_SH_SL_RT_FLT_GEN : INT  := 8;	//COKE SPILLAGE SHOVEL SLEW RETRACT FAULT GENERATION TIME
   CK_SPI_SH_SL_RT_OP_CT_T : INT ;	//COKE SPILLAGE SHOVEL SLEW RETRACT OUTPUT CUT TIMER
   CK_SPI_SH_SL_RT_FLT : BOOL ;	//COKE SPILLAGE SHOVEL SLEW RETRACT FAULT
   CK_SPI_SH_SL_AUTO_RT_OVR : BOOL ;	//COKE SPILLAGE SHOVEL SLEW AUTO RETRACT OVER
   CK_SPI_SH_SL_AUTO_RT_DEL : INT  := 3;	//COKE SPILLAGE SHOVEL SLEW AUTO RETRACT OVER DELAY
   CK_SPI_SH_SL_ATO_RT_DL_T : INT ;	//COKE SPILLAGE SHOVEL SLEW AUTO RETRACT OVER DELAY TIMER
   DR_CL_SH_SL_FW_OP_CUT : BOOL ;	//DOOR CLEANER SPILLAGE SHOVEL SLEW FORWARD OUTPUT CUT
   DR_CL_SH_SL_FW_FLT_TMR : INT ;	//DOOR CLEANER SPILLAGE SHOVEL SLEW FORWARD FAULT TIMER
   DR_CL_SH_SL_FW_FLT_GEN : INT  := 8;	//DOOR CLEANER SPILLAGE SHOVEL SLEW FORWARD FAULT GENERATION TIME
   DR_CL_SH_SL_FW_OP_CT_T : INT ;	//DOOR CLEANER SPILLAGE SHOVEL SLEW FORWARD OUTPUT CUT TIMER
   DR_CL_SH_SL_FW_FLT : BOOL ;	//DOOR CLEANER SPILLAGE SHOVEL SLEW FORWARD FAULT
   DR_CL_SH_SL_AUTO_FW_OVR : BOOL ;	//DOOR CLEANER SPILLAGE SHOVEL SLEW AUTO FORWARD OVER
   DR_CL_SH_SL_AUTO_FW_DEL : INT  := 3;	//DOOR CLEANER SPILLAGE SHOVEL SLEW AUTO FORWARD OVER DELAY
   DR_CL_SH_SL_ATO_FW_DL_T : INT ;	//DOOR CLEANER SPILLAGE SHOVEL SLEW AUTO FORWARD OVER DELAY TIMER
   DR_CL_SH_SL_RT_OP_CUT : BOOL ;	//DOOR CLEANER SPILLAGE SHOVEL SLEW RETRACT OUTPUT CUT
   DR_CL_SH_SL_RT_FLT_TMR : INT ;	//DOOR CLEANER SPILLAGE SHOVEL SLEW RETRACT FAULT TIMER
   DR_CL_SH_SL_RT_FLT_GEN : INT  := 8;	//DOOR CLEANER SPILLAGE SHOVEL SLEW RETRACT FAULT GENERATION TIME
   DR_CL_SH_SL_RT_OP_CT_T : INT ;	//DOOR CLEANER SPILLAGE SHOVEL SLEW RETRACT OUTPUT CUT TIMER
   DR_CL_SH_SL_RT_FLT : BOOL ;	//DOOR CLEANER SPILLAGE SHOVEL SLEW RETRACT FAULT
   DR_CL_SH_SL_AUTO_RT_OVR : BOOL ;	//DOOR CLEANER SPILLAGE SHOVEL SLEW AUTO RETRACT OVER
   DR_CL_SH_SL_AUTO_RT_DEL : INT  := 3;	//DOOR CLEANER SPILLAGE SHOVEL SLEW AUTO RETRACT OVER DELAY
   DR_CL_SH_SL_ATO_RT_DL_T : INT ;	//DOOR CLEANER SPILLAGE SHOVEL SLEW AUTO RETRACT OVER DELAY TIMER
   DR_CL_SP_HPR_FW_OP_CUT : BOOL ;	//DOOR CLEANER SPILLAGE HOPPER FORWARD OUTPUT CUT
   DR_CL_SP_HPR_FW_FLT_TMR : INT ;	//DOOR CLEANER SPILLAGE HOPPER FORWARD FAULT TIMER
   DR_CL_SP_HPR_FW_FLT_GEN : INT  := 8;	//DOOR CLEANER SPILLAGE HOPPER FORWARD FAULT GENERATION TIME
   DR_CL_SP_HPR_FW_OP_CT_T : INT ;	//DOOR CLEANER SPILLAGE HOPPER FORWARD OUTPUT CUT TIMER
   DR_CL_SP_HPR_FW_FLT : BOOL ;	//DOOR CLEANER SPILLAGE HOPPER FORWARD FAULT
   DR_CL_SP_HPR_AUTO_FW_OVR : BOOL ;	//DOOR CLEANER SPILLAGE HOPPER AUTO FORWARD OVER
   DR_CL_SP_HPR_AUTO_FW_DEL : INT  := 3;	//DOOR CLEANER SPILLAGE HOPPER AUTO FORWARD OVER DELAY
   DR_CL_SP_HPR_ATO_FW_DL_T : INT ;	//DOOR CLEANER SPILLAGE HOPPER AUTO FORWARD OVER DELAY TIMER
   DR_CL_SP_HPR_RT_OP_CUT : BOOL ;	//DOOR CLEANER SPILLAGE HOPPER RETRACT OUTPUT CUT
   DR_CL_SP_HPR_RT_FLT_TMR : INT ;	//DOOR CLEANER SPILLAGE HOPPER RETRACT FAULT TIMER
   DR_CL_SP_HPR_RT_FLT_GEN : INT  := 8;	//DOOR CLEANER SPILLAGE HOPPER RETRACT FAULT GENERATION TIME
   DR_CL_SP_HPR_RT_OP_CT_T : INT ;	//DOOR CLEANER SPILLAGE HOPPER RETRACT OUTPUT CUT TIMER
   DR_CL_SP_HPR_RT_FLT : BOOL ;	//DOOR CLEANER SPILLAGE HOPPER RETRACT FAULT
   DR_CL_SP_HPR_AUTO_RT_OVR : BOOL ;	//DOOR CLEANER SPILLAGE HOPPER AUTO RETRACT OVER
   DR_CL_SP_HPR_AUTO_RT_DEL : INT  := 3;	//DOOR CLEANER SPILLAGE HOPPER AUTO RETRACT OVER DELAY
   DR_CL_SP_HPR_ATO_RT_DL_T : INT ;	//DOOR CLEANER SPILLAGE HOPPER AUTO RETRACT OVER DELAY TIMER
   DR_CL_SP_HPR_FWD_STA_PB : BOOL ;	//DOOR CLEANER SPILLAGE HOPPER FORWARD START PUSH BUTTON
   DR_CL_SP_HPR_RET_STA_PB : BOOL ;	//DOOR CLEANER SPILLAGE HOPPER RETRACT START PUSH BUTTON
   DR_CL_SP_HPR_FWD_IND_LCS : BOOL ;	//DOOR CLEANER SPILLAGE HOPPER FORWARD INDICATOR LCS
   DR_CL_SP_HPR_RET_IND_LCS : BOOL ;	//DOOR CLEANER SPILLAGE HOPPER RETRACT INDICATOR LCS
  END_STRUCT ;	
BEGIN
   CL_SPI_CHT_DN_FLT_GEN := 8;
   CL_SPI_CHT_AUTO_DN_DEL := 3;
   CL_SPI_CHT_UP_FLT_GEN := 8;
   CL_SPI_CHT_AUTO_UP_DEL := 3;
   CL_SPI_HPR_GT_O_FLT_GEN := 8;
   CL_SPI_HPR_GT_AUTO_O_DEL := 3;
   CL_SPI_HPR_GT_C_FLT_GEN := 8;
   CL_SPI_HPR_GT_AUTO_C_DEL := 3;
   CK_SPI_SH_SL_FW_FLT_GEN := 8;
   CK_SPI_SH_SL_AUTO_FW_DEL := 3;
   CK_SPI_SH_SL_RT_FLT_GEN := 8;
   CK_SPI_SH_SL_AUTO_RT_DEL := 3;
   DR_CL_SH_SL_FW_FLT_GEN := 8;
   DR_CL_SH_SL_AUTO_FW_DEL := 3;
   DR_CL_SH_SL_RT_FLT_GEN := 8;
   DR_CL_SH_SL_AUTO_RT_DEL := 3;
   DR_CL_SP_HPR_FW_FLT_GEN := 8;
   DR_CL_SP_HPR_AUTO_FW_DEL := 3;
   DR_CL_SP_HPR_RT_FLT_GEN := 8;
   DR_CL_SP_HPR_AUTO_RT_DEL := 3;
END_DATA_BLOCK

DATA_BLOCK "TATA_COMMUNICATION_DB"	// DB 17
AUTHOR : Kamillas
VERSION : 0.1
  STRUCT
   TATA_DATA_READ_ERROR : INT ;	//TATA PLC DATA READ ERROR
   TATA_DATA_WRITE_ERROR : INT ;	//TATA PLC DATA WRITE ERROR
   PUSH_COMPLETED : BOOL ;	//PUSHING COMPLETED BIT
   LEV_COMPLETED : BOOL ;	//LEVELING COMPLETED BIT
   PUSH_COMP_LCH_TIMER : INT ;	//PUSHING COMPLETED BIT LATCH TIMER
   PUSH_COMP_LCH_TIME : INT  := 5;	//PUSHING COMPLETED BIT LATCH TIME
   LEV_COMP_LCH_TIMER : INT ;	//LEVELING COMPLETED BIT LATCH TIMER
   LEV_COMP_LCH_TIME : INT  := 5;	//LEVELING COMPLETED BIT LATCH TIME
   PUSLE_1 : BOOL ;	//PUSLE 1
   PUSLE_2 : BOOL ;	//PUSLE 2
   PUSLE_3 : BOOL ;	//PUSLE 3
   PUSLE_4 : BOOL ;	//PUSLE 4
   PUSLE_5 : BOOL ;	//PUSLE 5
   PUSLE_6 : BOOL ;	//PUSLE 6
   PUSLE_7 : BOOL ;	//PUSLE 7
   PUSLE_8 : BOOL ;	//PUSLE 8
   DR_OPN_LCH_TIMER : INT ;	//DOOR OPEN BIT LATCH TIMER
   DR_OPN_LCH_TIME : INT  := 5;	//DOOR OPEN BIT LATCH TIME
   DR_CLS_LCH_TIMER : INT ;	//DOOR CLOSE BIT LATCH TIMER
   DR_CLS_LCH_TIME : INT  := 5;	//DOOR CLOSE BIT LATCH TIME
   RAM_POS_DI : DINT ;	//RAM POSITION DOUBLE INTEGER
  END_STRUCT ;	
BEGIN
   PUSH_COMP_LCH_TIMER := 5;
   PUSH_COMP_LCH_TIME := 5;
   LEV_COMP_LCH_TIMER := 5;
   LEV_COMP_LCH_TIME := 5;
   DR_OPN_LCH_TIME := 5;
   DR_CLS_LCH_TIME := 5;
END_DATA_BLOCK

DATA_BLOCK "WINCC_DB"	// DB 18
AUTHOR : Kamillas
VERSION : 0.1
  STRUCT
   MAIN_PWR_ON_PB : BOOL ;	//MAIN POWER ON PUSH BUTTON
   MAIN_PWR_OFF_PB : BOOL ;	//MAIN POWER OFF PUSH BUTTON
   LAMP_TEST_PB : BOOL ;	//LAMP TEST PUSH BUTTON
   ALARM_ACK_PB : BOOL ;	//ALARM ACKNOWLEDGE PUSH BUTTON
   HYD_CD_LCS_SS : BOOL ;	//CONTROL DESK / LOCAL CONTROL SELECTOR SWITCH
   HYD_PUMP_1_2_SS : BOOL ;	//HYDRAULIC PUMP 1 OR 2 SELECTOR SWITCH
   HYD_PUMP_1_STA_PB : BOOL ;	//HYDRAULIC PUMP 1 START PUSH BUTTON
   HYD_PUMP_1_STP_PB : BOOL ;	//HYDRAULIC PUMP 1 STOP PUSH BUTTON
   HYD_PUMP_2_STA_PB : BOOL ;	//HYDRAULIC PUMP 2 START PUSH BUTTON
   HYD_PUMP_2_STP_PB : BOOL ;	//HYDRAULIC PUMP 2 STOP PUSH BUTTON
   AC_CD_LCS_SS : BOOL ;	//AIR COMPRESSOR CONTROL DESK/LOCAL CONTROL SELECTOR SWITCH
   AC_MTR_1_2_SS : BOOL ;	//AIR COMPRESSOR MOTOR 1/2 SELECTION
   AC_MTR_1_STA_PB : BOOL ;	//AIR COMPRESSOR MOTOR 1 START PUSH BUTTON
   AC_MTR_1_STP_PB : BOOL ;	//AIR COMPRESSOR MOTOR 1 STOP PUSH BUTTON
   AC_MTR_2_STA_PB : BOOL ;	//AIR COMPRESSOR MOTOR 2 START PUSH BUTTON
   AC_MTR_2_STP_PB : BOOL ;	//AIR COMPRESSOR MOTOR 2 STOP PUSH BUTTON
   LEV_DOOR_LOCAL_SS : BOOL ;	//LEVELER DOOR LOCAL SELECTOR SWITCH
   LEV_DOOR_MAN_SS : BOOL ;	//LEVELER DOOR MANUAL SELECTOR SWITCH
   LEV_DOOR_AUTO_SS : BOOL ;	//LEVELER DOOR AUTO SELECTOR SWITCH
   LEV_DOOR_STP_PB : BOOL  := TRUE;	//LEVELER DOOR STOP PUSH BUTTON
   ACT_GRP_FWD_STA_PB : BOOL ;	//LEVELER DOOR ACTUATING GRIP FORWARD START PUSH BUTTON
   ACT_GRP_RET_STA_PB : BOOL ;	//LEVELER DOOR ACTUATING GRIP RETRACT START PUSH BUTTON
   SLW_RK_SP_1_FWD_STA : BOOL ;	//LEVELER DOOR SLEAVING RACK STEP 1 FORWARD START PUSH BUTTON
   SLW_RK_SP_1_RET_STA : BOOL ;	//LEVELER DOOR SLEAVING RACK STEP 1 RETRACT START PUSH BUTTON
   SLW_RK_SP_2_FWD_STA : BOOL ;	//LEVELER DOOR SLEAVING RACK STEP 2 FORWARD START PUSH BUTTON
   SLW_RK_SP_2_RET_STA : BOOL ;	//LEVELER DOOR SLEAVING RACK STEP 2 RETRACT START PUSH BUTTON
   LEV_WN_CLR_UP_STA_PB : BOOL ;	//LEVELER DOOR LEVELER WINDOW FRAME CLEANER UP START PUSH BUTTON
   LEV_WN_CLR_DN_STA_PB : BOOL ;	//LEVELER DOOR LEVELER WINDOW FRAME CLEANER DOWN START PUSH BUTTON
   SMK_SLVE_FWD_STA_PB : BOOL ;	//LEVELER DOOR SMOKE SLEEVE FORWARD START PUSH BUTTON
   SMK_SLVE_RET_STA_PB : BOOL ;	//LEVELER DOOR SMOKE SLEEVE RETRACT START PUSH BUTTON
   LEV_BLOW_MTR_STA_PB : BOOL ;	//LEVELER BLOWER START PUSH BUTTON
   LEV_BLOW_MTR_STP_PB : BOOL ;	//LEVELER BLOWER STOP PUSH BUTTON
   CL_SPI_CHT_DN_STA : BOOL ;	//COAL SPILLAGE CHUTE DOWN START PUSH BUTTON
   CL_SPI_CHT_UP_STA : BOOL ;	//COAL SPILLAGE CHUTE UP START PUSH BUTTON
   PREP_DOOR_FUNC_STA : BOOL ;	//PREPARE DOOR FUNCTION START PUSH BUTTON
   PREP_DOOR_FUNC_STP : BOOL ;	//PREPARE DOOR FUNCTION STOP PUSH BUTTON
   FIN_DOOR_FUNC_STA : BOOL ;	//FINISH DOOR FUNCTION START PUSH BUTTON
   EXT_OVEN_DOR_AUTO_STA_PB : BOOL ;	//EXTRACT OVEN DOOR AUTO START PUSH BUTTON
   DR_EXT_RPL_AUTO_STP_PB : BOOL ;	//DOOR EXTRACTOR/REPLACE AUTO STOP PUSH BUTTON
   RPL_OVEN_DOR_AUTO_STA_PB : BOOL ;	//REPLACE OVEN DOOR AUTO START PUSH BUTTON
   CLEAN_OVN_DR_STA : BOOL ;	//CLEAN OVEN DOOR START PUSH BUTTON
   CLEAN_OVN_DR_STP : BOOL ;	//CLEAN OVEN DOOR STOP PUSH BUTTON
   PUSH_AUTO_STA_PB : BOOL ;	//PUSHER AUTO START PUSH BUTTON
   PUSH_AUTO_STP_RET_PB : BOOL ;	//PUSHER AUTO STOP AND RETRACT PUSH BUTTON
   PREP_FOR_LEV_STA_PB : BOOL ;	//PREPARE FOR LEVELLING START PUSH BUTTON
   PREP_FOR_LEV_STP_PB : BOOL ;	//PREPARE FOR LEVELLING STOP PUSH BUTTON
   FIN_LEV_DOOR_OPER_STA_PB : BOOL ;	//FINISH LEVELING DOOR OPERATIONS START PUSH BUTTON
   LEV_AUTO_STA_PB : BOOL ;	//LEVELER AUTO START PUSH BUTTON
   LEV_AUTO_STP_RET_PB : BOOL ;	//LEVELER AUTO STOP AND RETRACT PUSH BUTTON
   DOOR_CLNR_STP_PB : BOOL ;	//DOOR CLEANER STOP PUSH BUTTON
   CAR_TRA_FWD_STA_PB : BOOL ;	//CARRIAGE TRAVEL FORWARD START PUSH BUTTON
   CAR_TRA_RET_STA_PB : BOOL ;	//CARRIAGE TRAVEL RETRACT START PUSH BUTTON
   VER_CLNR_UP_STA_PB : BOOL ;	//VERTICAL CLEANER UP START PUSH BUTTON
   VER_CLNR_DN_STA_PB : BOOL ;	//VERTICAL CLEANER DOWN START PUSH BUTTON
   BTM_BRK_HLDR_UP_STA_PB : BOOL ;	//BOTTOM BRICK HOLDER FORWARD START PUSH BUTTON
   BTM_BRK_HLDR_DN_STA_PB : BOOL ;	//BOTTOM BRICK HOLDER RETRACT START PUSH BUTTON
   TOP_SCRP_FWD_STA_PB : BOOL ;	//TOP SCRAPPER FORWARD START PUSH BUTTON
   TOP_SCRP_RET_STA_PB : BOOL ;	//TOP SCRAPPER RETRACT START PUSH BUTTON
   BTM_SCRP_FWD_STA_PB : BOOL ;	//BOTTOM SCRAPPER FORWARD START PUSH BUTTON
   BTM_SCRP_RET_STA_PB : BOOL ;	//BOTTOM SCRAPPER RETRACT START PUSH BUTTON
   VIB_DOR_CLNR_STA_PB : BOOL ;	//VIBRATOR - DOOR CLEANER START PUSH BUTTON
   VIB_DOR_CLNR_STP_PB : BOOL ;	//VIBRATOR - DOOR CLEANER STOP PUSH BUTTON
   VIB_JMB_CLNR_STA_PB : BOOL ;	//VIBRATOR - JAMB CLEANER START PUSH BUTTON
   VIB_JMB_CLNR_STP_PB : BOOL ;	//VIBRATOR - JAMB CLEANER STOP PUSH BUTTON
   DC_SPI_SH_SL_FW_STA_PB : BOOL ;	//DOOR CLEANER SPILLAGE SHOVEL SLEW FORWARD START PUSH BUTTON
   DC_SPI_SH_SL_RT_STA_PB : BOOL ;	//DOOR CLEANER SPILLAGE SHOVEL SLEW RETRACT START PUSH BUTTON
   SLEW_FWD_STA_PB : BOOL ;	//SLEW FORWARD START PUSH BUTTON
   SLEW_RET_STA_PB : BOOL ;	//SLEW RETRACT START PUSH BUTTON
   TRA_FWD_STA_PB : BOOL ;	//TRAVEL FORWARD START PUSH BUTTON
   TRA_RET_STA_PB : BOOL ;	//TRAVEL RETRACT START PUSH BUTTON
   JC_VER_CLNR_UP_STA_PB : BOOL ;	//JAMP CLEANER VERTICAL CLEANER UP  START PUSH BUTTON
   JC_VER_CLNR_DN_STA_PB : BOOL ;	//JAMP CLEANER VERTICAL CLEANER DN START PUSH BUTTON
   JC_STOP_PB : BOOL ;	//JAMP CLEANER STOP PUSH BUTTON
   CNT_TH_WED_STOP_PB : BOOL ;	//COUNTER THRUST WEDGE STOP PUSH BUTTON
   CNT_TH_WED_UP_STA_PB : BOOL ;	//COUNTER THRUST WEDGE UP START PUSH BUTTON
   CNT_TH_WED_DN_STA_PB : BOOL ;	//COUNTER THRUST WEDGE DN START PUSH BUTTON
   PUSH_RAM_STP_PB : BOOL ;	//PUSHER RAM STOP PUSH BUTTON
   DOOR_EXT_STP_PB : BOOL ;	//DOOR EXTRACTOR STOP PUSH BUTTON
   DE_SLEW_FWD_STA_PB : BOOL ;	//SLEW FORWARD START PUSH BUTTON
   DE_SLEW_RET_STA_PB : BOOL ;	//SLEW RETRACT START
   VER_COMP_FWD_STA_PB : BOOL ;	//VERTICAL COMPENSATION FORWARD START PUSH BUTTON
   VER_COMP_RET_STA_PB : BOOL ;	//VERTICAL COMPENSATION RETRACT START PUSH BUTTON
   DE_TRA_FWD_STA_PB : BOOL ;	//TRAVEL FORWARD START PUSH BUTTON
   DE_TRA_RET_STA_PB : BOOL ;	//TRAVEL RETRACT START PUSH BUTTON
   MAIN_STK_UP_STA_PB : BOOL ;	//MAIN STROKE UP START PUSH BUTTON
   MAIN_STK_UP_DN_PB : BOOL ;	//MAIN STROKE DOWN START PUSH BUTTON
   FIN_STK_UP_STA_PB : BOOL ;	//FINAL STROKE UP START PUSH BUTTON
   FIN_STK_UP_DN_PB : BOOL ;	//FINAL STROKE DOWN START PUSH BUTTON
   PRE_STK_UP_STA_PB : BOOL ;	//PRE STROKE UP START PUSH BUTTON
   PRE_STK_UP_DN_PB : BOOL ;	//PRE STROKE DOWN START PUSH BUTTON
   DR_SPNG_LK_STA_PB : BOOL ;	//DOOR SPRING PRESSURE START PUSH BUTTON
   DR_SPNG_UNLK_STA_PB : BOOL ;	//DOOR SPRING PRESSURE RELEASE START PUSH BUTTON
   DR_LCH_TURN_UP_PB : BOOL ;	//DOOR LATCH TURNING LOCK PUSH BUTTON
   DR_LCH_TURN_DN_PB : BOOL ;	//DOOR LATCH TURNING UNLOCK PUSH BUTTON
   NO_USE : BOOL ;
   NO_USE1 : BOOL ;
   OPER_MODE_SS : BOOL ;
   NO_USE2 : BOOL ;
   NO_USE3 : BOOL ;
   NO_USE4 : BOOL ;
   NO_USE5 : BOOL ;
   NO_USE6 : BOOL ;
   NO_USE7 : BOOL ;
   NO_USE8 : BOOL ;
   HYD_PUMP_CD_LCS : BOOL ;
   NO_USE9 : BOOL ;
   NO_USE10 : BOOL ;
   NO_USE11 : BOOL ;
   NO_USE12 : BOOL ;
   NO_USE13 : BOOL ;
   NO_USE14 : BOOL ;
   NO_USE15 : BOOL ;
   PUMP_1_2_SS : BOOL ;
   NO_USE16 : BOOL ;
   NO_USE17 : BOOL ;
   NO_USE18 : BOOL ;
   NO_USE19 : BOOL ;
   NO_USE20 : BOOL ;
   NO_USE21 : BOOL ;
   NO_USE22 : BOOL ;
   AIR_COMP_CD_LCS_SS : BOOL ;
   NO_USE23 : BOOL ;
   NO_USE24 : BOOL ;
   NO_USE25 : BOOL ;
   NO_USE26 : BOOL ;
   NO_USE27 : BOOL ;
   NO_USE28 : BOOL ;
   NO_USE29 : BOOL ;
   AIR_COMP_MTR_1_2_SS : BOOL ;
   NO_USE30 : BOOL ;
   NO_USE31 : BOOL ;
   NO_USE32 : BOOL ;
   NO_USE33 : BOOL ;
   NO_USE34 : BOOL ;
   NO_USE35 : BOOL ;
   NO_USE36 : BOOL ;
   LEVELLER_SELEC : BOOL ;
   NO_USE37 : BOOL ;
   NO_USE38 : BOOL ;
   NO_USE39 : BOOL ;
   NO_USE40 : BOOL ;
   NO_USE41 : BOOL ;
   NO_USE42 : BOOL ;
   NO_USE43 : BOOL ;
   LEV_IN_MAN_MODE : BOOL ;
   LEV_IN_AUTO_MODE : BOOL ;
   NO_USE44 : BOOL ;
   NO_USE45 : BOOL ;
   NO_USE46 : BOOL ;
   NO_USE47 : BOOL ;
   NO_USE48 : BOOL ;
   NO_USE49 : BOOL ;
   REPAIR_MODE_SS : BOOL ;
   NO_USE50 : BOOL ;
   NO_USE51 : BOOL ;
   NO_USE52 : BOOL ;
   NO_USE53 : BOOL ;
   NO_USE54 : BOOL ;
   NO_USE55 : BOOL ;
   NO_USE56 : BOOL ;
   DC_AUTO_MAN_SS : BOOL ;
   NO_USE57 : BOOL ;
   NO_USE58 : BOOL ;
   NO_USE59 : BOOL ;
   NO_USE60 : BOOL ;
   NO_USE61 : BOOL ;
   NO_USE62 : BOOL ;
   NO_USE63 : BOOL ;
   DC_AUTO_SS : BOOL ;
   DC_MAN_SS : BOOL ;
   NO_USE64 : BOOL ;
   NO_USE65 : BOOL ;
   NO_USE66 : BOOL ;
   NO_USE67 : BOOL ;
   NO_USE68 : BOOL ;
   NO_USE69 : BOOL ;
   OPER_RM_SS : BOOL ;
   NO_USE70 : BOOL ;
   NO_USE71 : BOOL ;
   NO_USE72 : BOOL ;
   NO_USE73 : BOOL ;
   NO_USE74 : BOOL ;
   NO_USE75 : BOOL ;
   NO_USE76 : BOOL ;
   TRAV_AUTO_MAN_SS : BOOL ;
   NO_USE77 : BOOL ;
   NO_USE78 : BOOL ;
   NO_USE79 : BOOL ;
   NO_USE80 : BOOL ;
   NO_USE81 : BOOL ;
   NO_USE82 : BOOL ;
   NO_USE83 : BOOL ;
   TRAVEL_AUTO_MAN_SS_TAG : BOOL ;
   NO_USE84 : BOOL ;
   NO_USE85 : BOOL ;
   NO_USE86 : BOOL ;
   NO_USE87 : BOOL ;
   NO_USE88 : BOOL ;
   NO_USE89 : BOOL ;
   NO_USE90 : BOOL ;
   LEV_RAM_AUTO_SS : BOOL ;
   LEV_RAM_MAN_SS : BOOL ;
   LEVE_RAM_STP_PB : BOOL ;
   NO_USE93 : BOOL ;
   NO_USE94 : BOOL ;
   NO_USE95 : BOOL ;
   NO_USE96 : BOOL ;
   NO_USE97 : BOOL ;
   JC_AUTO_MAN_SS_TAG : BOOL ;
   NO_USE98 : BOOL ;
   NO_USE99 : BOOL ;
   NO_USE100 : BOOL ;
   NO_USE101 : BOOL ;
   NO_USE102 : BOOL ;
   NO_USE103 : BOOL ;
   NO_USE104 : BOOL ;
   LEVE_RAM_AUTO_MAN_SS_TAG : BOOL ;
   NO_USE105 : BOOL ;
   NO_USE106 : BOOL ;
   NO_USE107 : BOOL ;
   NO_USE108 : BOOL ;
   NO_USE109 : BOOL ;
   NO_USE110 : BOOL ;
   NO_USE111 : BOOL ;
   JC_AUTO_SS : BOOL ;
   JC_MAN_SS : BOOL ;
   CNT_TH_WED_MAN_SS : BOOL ;
   CNT_TH_WED_AUTO_SS : BOOL ;
   PUSHER_MAN_SS : BOOL ;
   PUSHER_AUTO_SS : BOOL ;
   DE_AUTO_SS : BOOL ;
   DE_MAN_SS : BOOL ;
   CNT_THRST_AUTO_MAN_SS : BOOL ;
   NO_USE91 : BOOL ;
   NO_USE92 : BOOL ;
   NO_USE114 : BOOL ;
   NO_USE115 : BOOL ;
   NO_USE116 : BOOL ;
   NO_USE117 : BOOL ;
   NO_USE118 : BOOL ;
   PUSHER_AUTO_MAN_SS_TAG : BOOL ;
   NO_USE112 : BOOL ;
   NO_USE113 : BOOL ;
   NO_USE119 : BOOL ;
   NO_USE120 : BOOL ;
   NO_USE121 : BOOL ;
   NO_USE122 : BOOL ;
   NO_USE123 : BOOL ;
   DE_AUTO_MAN_SS_TAG : BOOL ;
   NO_USE124 : BOOL ;
   NO_USE125 : BOOL ;
   NO_USE126 : BOOL ;
   NO_USE127 : BOOL ;
   NO_USE128 : BOOL ;
   NO_USE129 : BOOL ;
   NO_USE130 : BOOL ;
   DE_STP_PB : BOOL ;
   GRV_SCRP_FWD_PB : BOOL ;
   GRV_SCRP_RET_PB : BOOL ;
   CK_SPI_SH_SL_FW_STA_PB : BOOL ;
   CK_SPI_SH_SL_RET_STA_PB : BOOL ;
   CLN_OVN_JMB_AUTO_STA_PB : BOOL ;
   CLN_OVN_JMB_AUTO_STP_PB : BOOL ;
   EMER_STP_PB : BOOL ;
   SIR_ON_PB : BOOL ;
  END_STRUCT ;	
BEGIN
   MAIN_PWR_OFF_PB := TRUE;
   HYD_PUMP_1_STP_PB := TRUE;
   HYD_PUMP_2_STP_PB := TRUE;
   AC_MTR_1_STP_PB := TRUE;
   AC_MTR_2_STP_PB := TRUE;
   LEV_DOOR_STP_PB := TRUE;
   LEV_BLOW_MTR_STP_PB := TRUE;
   PREP_DOOR_FUNC_STP := TRUE;
   DR_EXT_RPL_AUTO_STP_PB := TRUE;
   CLEAN_OVN_DR_STP := TRUE;
   PUSH_AUTO_STP_RET_PB := TRUE;
   PREP_FOR_LEV_STP_PB := TRUE;
   LEV_AUTO_STP_RET_PB := TRUE;
   DOOR_CLNR_STP_PB := TRUE;
   VIB_DOR_CLNR_STP_PB := TRUE;
   VIB_JMB_CLNR_STP_PB := TRUE;
   JC_STOP_PB := TRUE;
   CNT_TH_WED_STOP_PB := TRUE;
   PUSH_RAM_STP_PB := TRUE;
   DOOR_EXT_STP_PB := TRUE;
   LEVE_RAM_STP_PB := TRUE;
   DE_STP_PB := TRUE;
   CLN_OVN_JMB_AUTO_STP_PB := TRUE;
END_DATA_BLOCK

DATA_BLOCK "DB_FOR_FM350"	// DB 19
AUTHOR : Kamillas
VERSION : 0.1
  STRUCT
   JOB_WR : STRUCT 	// write commands
    NO : BYTE ;	// number
    BUSY : BOOL ;	// job in working
    DONE : BOOL ;	// job is done
    IMPOSS : BOOL ;	// job impossible
    UNKOWN : BOOL ;	// job unkown
   END_STRUCT ;
   JOB_RD : STRUCT 	// read commands
    NO : BYTE ;	// number
    BUSY : BOOL ;	// job in working
    DONE : BOOL ;	// job is done
    IMPOSS : BOOL ;	// job impossible
    UNKOWN : BOOL ;	// job unkown
   END_STRUCT ;
   RESERV_0 : ARRAY  [1 .. 3 ] OF WORD  := 3 (W#16#0) ;	// reserved
   RESERV_1 : WORD ;	// reserved
   MOD_ADR : WORD ;	// module address
   CH_ADR : DWORD ;	// channel address
   DS_OFFS : BYTE ;	// data block offset
   RESERV_2 : BYTE ;	// reserved
   CONTROL_SIGNALS : STRUCT 	// control signals
    BIT0_0 : BOOL ;	// reserved
    BIT0_1 : BOOL ;	// reserved
    BIT0_2 : BOOL ;	// reserved
    BIT0_3 : BOOL ;	// reserved
    BIT0_4 : BOOL ;	// reserved
    BIT0_5 : BOOL ;	// reserved
    BIT0_6 : BOOL ;	// reserved
    BIT0_7 : BOOL ;	// reserved
    CTRL_DQ0 : BOOL ;	// control digital output DQ0
    CTRL_DQ1 : BOOL ;	// control digital output DQ1
    CTRL_DQ2 : BOOL ;	// control digital output DQ2
    CTRL_DQ3 : BOOL ;	// control digital output DQ3
    CTRL_DQ4 : BOOL ;	// control digital output DQ4
    CTRL_DQ5 : BOOL ;	// control digital output DQ5
    CTRL_DQ6 : BOOL ;	// control digital output DQ6
    CTRL_DQ7 : BOOL ;	// control digital output DQ7
    SET_DQ0 : BOOL ;	// set digital output DQ0
    SET_DQ1 : BOOL ;	// set digital output DQ1
    SET_DQ2 : BOOL ;	// set digital output DQ2
    SET_DQ3 : BOOL ;	// set digital output DQ3
    SET_DQ4 : BOOL ;	// set digital output DQ4
    SET_DQ5 : BOOL ;	// set digital output DQ5
    SET_DQ6 : BOOL ;	// set digital output DQ6
    SET_DQ7 : BOOL ;	// set digital output DQ7
    SW_GATE0 : BOOL ;	// software gate 0
    SW_GATE1 : BOOL ;	// software gate 1
    SW_GATE2 : BOOL ;	// software gate 2
    SW_GATE3 : BOOL ;	// software gate 3
    SW_GATE4 : BOOL ;	// software gate 4
    SW_GATE5 : BOOL ;	// software gate 5
    SW_GATE6 : BOOL ;	// software gate 6
    SW_GATE7 : BOOL ;	// software gate 7
    CTRL_DWORD1 : DWORD ;	// reserved
    CTRL_DWORD2 : DWORD ;	// reserved
    CTRL_DWORD3 : DWORD ;	// reserved
   END_STRUCT ;
   CHECKBACK_SIGNALS : STRUCT 	// checkback signals
    BIT0_0 : BOOL ;	// reserved
    STS_TFB : BOOL ;	// status test free bit
    BIT0_2 : BOOL ;	// reserved
    BIT0_3 : BOOL ;	// reserved
    DATA_ERR : BOOL ;	// data error bit
    BIT0_5 : BOOL ;	// reserved
    BIT0_6 : BOOL ;	// reserved
    PARA : BOOL ;	// module parametrized
    STS_CMP0 : BOOL ;	// status compare event 0
    STS_CMP1 : BOOL ;	// status compare event 1
    STS_CMP2 : BOOL ;	// status compare event 2
    STS_CMP3 : BOOL ;	// status compare event 3
    STS_CMP4 : BOOL ;	// status compare event 4
    STS_CMP5 : BOOL ;	// status compare event 5
    STS_CMP6 : BOOL ;	// status compare event 6
    STS_CMP7 : BOOL ;	// status compare event 7
    STS_UFLW0 : BOOL ;	// status counter 0 passed the underflow value
    STS_UFLW1 : BOOL ;	// status counter 1 passed the underflow value
    STS_UFLW2 : BOOL ;	// status counter 2 passed the underflow value
    STS_UFLW3 : BOOL ;	// status counter 3 passed the underflow value
    STS_UFLW4 : BOOL ;	// status counter 4 passed the underflow value
    STS_UFLW5 : BOOL ;	// status counter 5 passed the underflow value
    STS_UFLW6 : BOOL ;	// status counter 6 passed the underflow value
    STS_UFLW7 : BOOL ;	// status counter 7 passed the underflow value
    STS_OFLW0 : BOOL ;	// status counter 0 passed the overflow value
    STS_OFLW1 : BOOL ;	// status counter 1 passed the overflow value
    STS_OFLW2 : BOOL ;	// status counter 2 passed the overflow value
    STS_OFLW3 : BOOL ;	// status counter 3 passed the overflow value
    STS_OFLW4 : BOOL ;	// status counter 4 passed the overflow value
    STS_OFLW5 : BOOL ;	// status counter 5 passed the overflow value
    STS_OFLW6 : BOOL ;	// status counter 6 passed the overflow value
    STS_OFLW7 : BOOL ;	// status counter 7 passed the overflow value
    STS_DIR0 : BOOL ;	// status counter 0 direction
    STS_DIR1 : BOOL ;	// status counter 1 direction
    STS_DIR2 : BOOL ;	// status counter 2 direction
    STS_DIR3 : BOOL ;	// status counter 3 direction
    STS_DIR4 : BOOL ;	// status counter 4 direction
    STS_DIR5 : BOOL ;	// status counter 5 direction
    STS_DIR6 : BOOL ;	// status counter 6 direction
    STS_DIR7 : BOOL ;	// status counter 7 direction
    STS_DI0 : BOOL ;	// status of the digital input 0
    STS_DI1 : BOOL ;	// status of the digital input 1
    STS_DI2 : BOOL ;	// status of the digital input 2
    STS_DI3 : BOOL ;	// status of the digital input 3
    STS_DI4 : BOOL ;	// status of the digital input 4
    STS_DI5 : BOOL ;	// status of the digital input 5
    STS_DI6 : BOOL ;	// status of the digital input 6
    STS_DI7 : BOOL ;	// status of the digital input 7
    STS_DQ0 : BOOL ;	// status of the digital output 0
    STS_DQ1 : BOOL ;	// status of the digital output 1
    STS_DQ2 : BOOL ;	// status of the digital output 2
    STS_DQ3 : BOOL ;	// status of the digital output 3
    STS_DQ4 : BOOL ;	// status of the digital output 4
    STS_DQ5 : BOOL ;	// status of the digital output 5
    STS_DQ6 : BOOL ;	// status of the digital output 6
    STS_DQ7 : BOOL ;	// status of the digital output 7
    STS_GATE0 : BOOL ;	// status of the internal gate 0
    STS_GATE1 : BOOL ;	// status of the internal gate 1
    STS_GATE2 : BOOL ;	// status of the internal gate 2
    STS_GATE3 : BOOL ;	// status of the internal gate 3
    STS_GATE4 : BOOL ;	// status of the internal gate 4
    STS_GATE5 : BOOL ;	// status of the internal gate 5
    STS_GATE6 : BOOL ;	// status of the internal gate 6
    STS_GATE7 : BOOL ;	// status of the internal gate 7
    USER_STAT_WORD0 : WORD ;	// user specific status
    USER_STAT_WORD1 : WORD ;	// user specific status
    USER_STAT_WORD2 : WORD ;	// user specific status
    USER_STAT_WORD3 : WORD ;	// user specific status
   END_STRUCT ;
   LOAD_VAL0 : DINT ;	// load value counter 0
   LOAD_VAL1 : DINT ;	// load value counter 1
   LOAD_VAL2 : DINT ;	// load value counter 2
   LOAD_VAL3 : DINT ;	// load value counter 3
   LOAD_VAL4 : DINT ;	// load value counter 4
   LOAD_VAL5 : DINT ;	// load value counter 5
   LOAD_VAL6 : DINT ;	// load value counter 6
   LOAD_VAL7 : DINT ;	// load value counter 7
   LOAD_PREPARE_VAL0 : DINT ;	// load prepare value counter 0
   LOAD_PREPARE_VAL1 : DINT ;	// load prepare value counter 1
   LOAD_PREPARE_VAL2 : DINT ;	// load prepare value counter 2
   LOAD_PREPARE_VAL3 : DINT ;	// load prepare value counter 3
   LOAD_PREPARE_VAL4 : DINT ;	// load prepare value counter 4
   LOAD_PREPARE_VAL5 : DINT ;	// load prepare value counter 5
   LOAD_PREPARE_VAL6 : DINT ;	// load prepare value counter 6
   LOAD_PREPARE_VAL7 : DINT ;	// load prepare value counter 7
   CMP_VAL0 : DINT ;	// comparator value 0
   CMP_VAL1 : DINT ;	// comparator value 1
   CMP_VAL2 : DINT ;	// comparator value 2
   CMP_VAL3 : DINT ;	// comparator value 3
   CMP_VAL4 : DINT ;	// comparator value 4
   CMP_VAL5 : DINT ;	// comparator value 5
   CMP_VAL6 : DINT ;	// comparator value 6
   CMP_VAL7 : DINT ;	// comparator value 7
   ACT_CNTV0 : DINT ;	// actual counter value 0
   ACT_MSRV0 : DINT ;	// act. measurement value 0
   ACT_CNTV1 : DINT ;	// actual counter value 1
   ACT_MSRV1 : DINT ;	// act. measurement value 1
   ACT_CNTV2 : DINT ;	// actual counter value 2
   ACT_MSRV2 : DINT ;	// act. measurement value 2
   ACT_CNTV3 : DINT ;	// actual counter value 3
   ACT_MSRV3 : DINT ;	// act. measurement value 3
   ACT_CNTV4 : DINT ;	// actual counter value 4
   ACT_MSRV4 : DINT ;	// act. measurement value 4
   ACT_CNTV5 : DINT ;	// actual counter value 5
   ACT_MSRV5 : DINT ;	// act. measurement value 5
   ACT_CNTV6 : DINT ;	// actual counter value 6
   ACT_MSRV6 : DINT ;	// act. measurement value 6
   ACT_CNTV7 : DINT ;	// actual counter value 7
   ACT_MSRV7 : DINT ;	// act. measurement value 7
   DIAGNOSTIC_INT_INFO : STRUCT 	// diagnostic int. information
    BYTE0 : BYTE ;	// byte 0
    BYTE1 : BYTE ;	// byte 1
    BYTE2 : BYTE ;	// byte 2
    BYTE3 : BYTE ;	// byte 3
    BYTE4 : BYTE ;	// channel type info
    BYTE5 : BYTE ;	// channel info length
    BYTE6 : BYTE ;	// number of channels
    BYTE7 : BYTE ;	// channel error vector
    BYTE8 : BYTE ;	// error counter 0
    BYTE9 : BYTE ;	// error counter 1
    BYTE10 : BYTE ;	// error counter 2
    BYTE11 : BYTE ;	// error counter 3
    BYTE12 : BYTE ;	// error counter 4
    BYTE13 : BYTE ;	// error counter 5
    BYTE14 : BYTE ;	// error counter 6
    BYTE15 : BYTE ;	// error counter 7
   END_STRUCT ;
  END_STRUCT ;	
BEGIN
   MOD_ADR := W#16#110;
   CH_ADR := DW#16#880;
END_DATA_BLOCK

DATA_BLOCK "FB_TO_TATA"	// DB 20
AUTHOR : Kamillas
VERSION : 0.1
  STRUCT
   PC_MACHINE_STATUS_BIT : STRUCT
    PC_PUSH_START : BOOL ;	//Pushing started
    PC_PUSH_COMPLET : BOOL ;	//Pushing completed
    PC_STATU : BOOL ;	//Status of pusher
    PC_RAM_FWD : BOOL ;	//Permissive for allowing the Ram to move fwd
    PC_STRT_LEVLING : BOOL ;	//Confirming start of leveling
    PC_STOP_LEVLING : BOOL ;	//Confirming end of leveling
    PC_PUSH_SIDE_DOOR_CL : BOOL ;	//Door open
    PC_PUSH_SIDE_DOOR_OP : BOOL ;	//Door close
    PC_DRV_STATU : BOOL ;	//Drive healthy/unhealthy
    PC_DRV_FWD : BOOL ;	//Motion towards quenching tower
    PC_DRV_REV : BOOL ;	//Motion towards coal tower
    PC_RAM_OVN_FAC_RCHD : BOOL ;	//PUSHER RAM OVEN FACE REACHED
    PC_RAM_FWD_END_RCHD : BOOL ;	//PUSHER RAM FORWARD END REACHED
    PC_TRA_MODE : BOOL ;	//PUSHER CAR TRAVEL MODE
    PC_GUIDE_CAGE_ENTRY : BOOL ;	//PUSHER RAM REACHED AT GUIDE CAGE ENTRY
    PC_HOOD_ON_CMD : BOOL ;	//HOOD ON COMMAND
    PC_PUSH_SPEED : REAL ;	//Pusher speed feedback
    PC_PUSH_CURRENT : INT ;	//Pusher current
    PC_RAM_POS : REAL ;	//Pusher Ram position
    PC_LEVL_CURRENT : INT ;	//LEVELER BAR DRIVE CURRENT
    SATA : ARRAY  [1 .. 2 ] OF INT ;
   END_STRUCT ;
  END_STRUCT ;	
BEGIN
END_DATA_BLOCK

DATA_BLOCK "CMD_FROM_TATA"	// DB 21
AUTHOR : Kamillas
VERSION : 0.1
  STRUCT
   PC_OnBord_STATUS_BIT : STRUCT
    PC_PUSH_PERM : BOOL ;	//Pushing interlock OK
    PC_PUSH_LT_MODE : BOOL ;	//Long travel in auto or in man
    PC_TRAVEL_FWD : BOOL ;	//FWD over profibus
    PC_TRAVEL_REV : BOOL ;	//REV over profibus
    PC_TRAVEL_START : BOOL ;	//START over profibus
    PC_TRAVEL_STOP : BOOL ;	//STOP  over profibus
    SpareBit_1 : BOOL ;
    SpareBit_2 : BOOL ;
    SpareBit_3 : BOOL ;
    SpareBit_4 : BOOL ;
    SpareBit_5 : BOOL ;
    SpareBit_6 : BOOL ;
    SpareBit_7 : BOOL ;
    SpareBit_8 : BOOL ;
    SpareBit_9 : BOOL ;
    SpareBit_10 : BOOL ;
    PC_SPEED_REF : INT ;	//Reserve for LT motion (spd_ref) over profibus
    SATA : ARRAY  [1 .. 7 ] OF INT ;
   END_STRUCT ;
  END_STRUCT ;	
BEGIN
END_DATA_BLOCK

ORGANIZATION_BLOCK "MAIN_PROGRAM"	// OB 1
AUTHOR : Kamillas
VERSION : 0.1
BEGIN
// (block stored without names or comments; labels and parameter names are numbered)
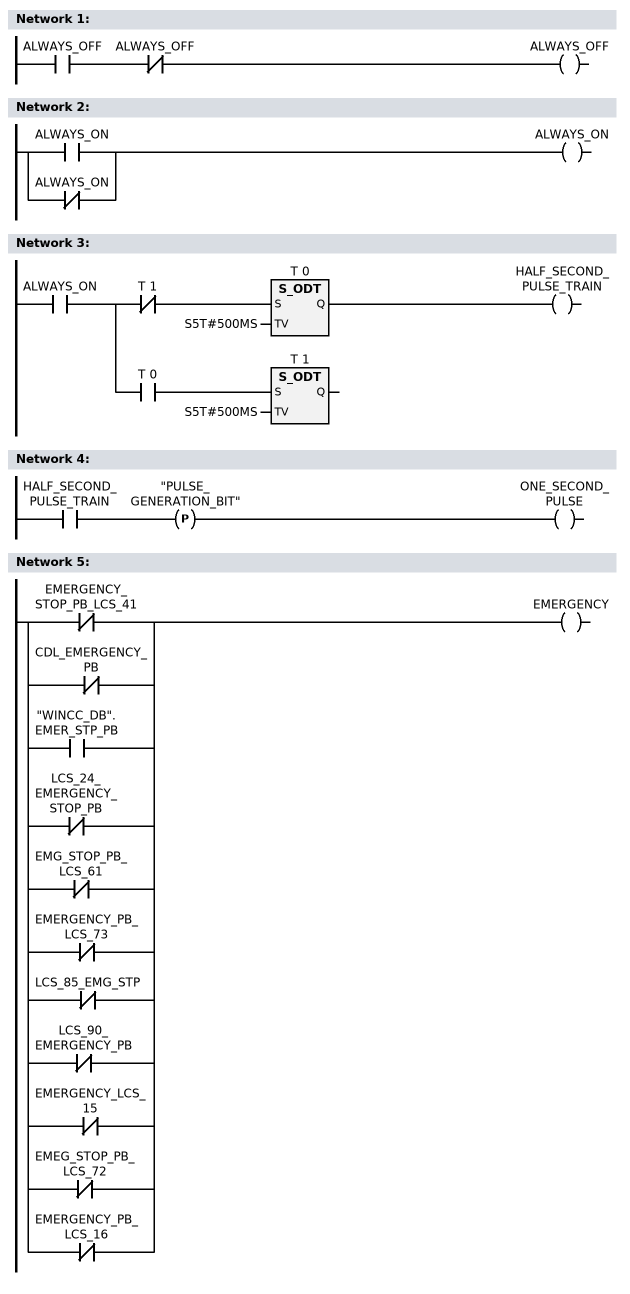
NETWORK
TITLE =
      A     "ALWAYS_OFF";
      AN    "ALWAYS_OFF";
      =     "ALWAYS_OFF";
NETWORK
TITLE =
      O     "ALWAYS_ON";
      ON    "ALWAYS_ON";
      =     "ALWAYS_ON";
NETWORK
TITLE =
      A     "ALWAYS_ON";
      =     L 20.0;
      A     L 20.0;
      AN    T 1;
      L     S5T#500MS;
      SD    T 0;
      NOP   0;
      NOP   0;
      NOP   0;
      A     T 0;
      =     "HALF_SECOND_PULSE_TRAIN";
      A     L 20.0;
      A     T 0;
      L     S5T#500MS;
      SD    T 1;
      NOP   0;
      NOP   0;
      NOP   0;
      NOP   0;
NETWORK
TITLE =
      A     "HALF_SECOND_PULSE_TRAIN";
      FP    "PULSE_GENERATION_BIT";
      =     "ONE_SECOND_PULSE";
NETWORK
TITLE =
      ON    "EMERGENCY_STOP_PB_LCS_41";
      ON    "CDL_EMERGENCY_PB";
      O     "WINCC_DB".EMER_STP_PB;
      ON    "LCS_24_EMERGENCY_STOP_PB";
      ON    "EMG_STOP_PB_LCS_61";
      ON    "EMERGENCY_PB_LCS_73";
      ON    "LCS_85_EMG_STP";
      ON    "LCS_90_EMERGENCY_PB";
      ON    "EMERGENCY_LCS_15";
      ON    "EMEG_STOP_PB_LCS_72";
      ON    "EMERGENCY_PB_LCS_16";
      =     "EMERGENCY";
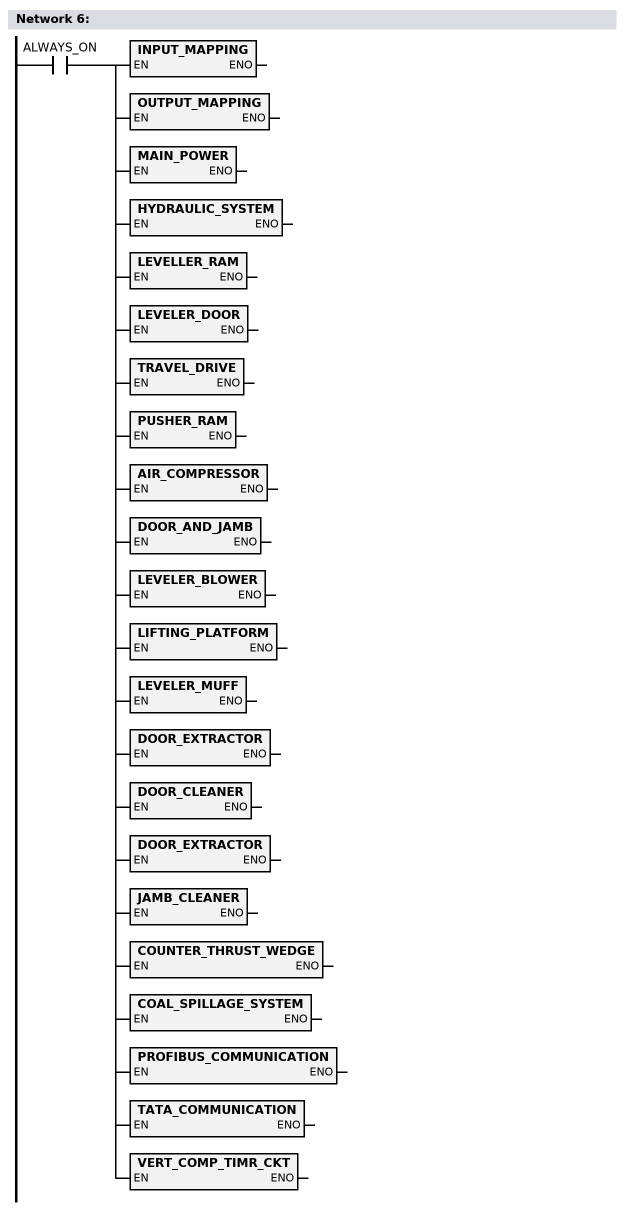
NETWORK
TITLE =
      A     "ALWAYS_ON";
      =     L 20.0;
      A     L 20.0;
      JNB   M001;
      CALL  "INPUT_MAPPING";
M001: NOP   0;
      A     L 20.0;
      JNB   M002;
      CALL  "OUTPUT_MAPPING";
M002: NOP   0;
      A     L 20.0;
      JNB   M003;
      CALL  "MAIN_POWER";
M003: NOP   0;
      A     L 20.0;
      JNB   M004;
      CALL  "HYDRAULIC_SYSTEM";
M004: NOP   0;
      A     L 20.0;
      JNB   M005;
      CALL  "LEVELLER_RAM";
M005: NOP   0;
      A     L 20.0;
      JNB   M006;
      CALL  "LEVELER_DOOR";
M006: NOP   0;
      A     L 20.0;
      JNB   M007;
      CALL  "TRAVEL_DRIVE";
M007: NOP   0;
      A     L 20.0;
      JNB   M008;
      CALL  "PUSHER_RAM";
M008: NOP   0;
      A     L 20.0;
      JNB   M009;
      CALL  "AIR_COMPRESSOR";
M009: NOP   0;
      A     L 20.0;
      JNB   M010;
      CALL  "DOOR_AND_JAMB";
M010: NOP   0;
      A     L 20.0;
      JNB   M011;
      CALL  "LEVELER_BLOWER";
M011: NOP   0;
      A     L 20.0;
      JNB   M012;
      CALL  "LIFTING_PLATFORM";
M012: NOP   0;
      A     L 20.0;
      JNB   M013;
      CALL  "LEVELER_MUFF";
M013: NOP   0;
      A     L 20.0;
      JNB   M014;
      CALL  "DOOR_EXTRACTOR";
M014: NOP   0;
      A     L 20.0;
      JNB   M015;
      CALL  "DOOR_CLEANER";
M015: NOP   0;
      A     L 20.0;
      JNB   M016;
      CALL  "DOOR_EXTRACTOR";
M016: NOP   0;
      A     L 20.0;
      JNB   M017;
      CALL  "JAMB_CLEANER";
M017: NOP   0;
      A     L 20.0;
      JNB   M018;
      CALL  "COUNTER_THRUST_WEDGE";
M018: NOP   0;
      A     L 20.0;
      JNB   M019;
      CALL  "COAL_SPILLAGE_SYSTEM";
M019: NOP   0;
      A     L 20.0;
      JNB   M020;
      CALL  "PROFIBUS_COMMUNICATION";
M020: NOP   0;
      A     L 20.0;
      JNB   M021;
      CALL  "TATA_COMMUNICATION";
M021: NOP   0;
      A     L 20.0;
      JNB   M022;
      CALL  "VERT_COMP_TIMR_CKT";
M022: NOP   0;
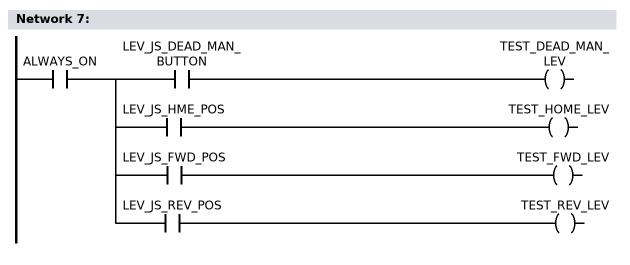
NETWORK
TITLE =
      A     "ALWAYS_ON";
      =     L 20.0;
      A     L 20.0;
      A     "LEV_JS_DEAD_MAN_BUTTON";
      =     "TEST_DEAD_MAN_LEV";
      A     L 20.0;
      A     "LEV_JS_HME_POS";
      =     "TEST_HOME_LEV";
      A     L 20.0;
      A     "LEV_JS_FWD_POS";
      =     "TEST_FWD_LEV";
      A     L 20.0;
      A     "LEV_JS_REV_POS";
      =     "TEST_REV_LEV";
END_ORGANIZATION_BLOCK

ORGANIZATION_BLOCK "I/O_FLT1"	// OB 82
AUTHOR : Kamillas
VERSION : 0.1
BEGIN
// (block stored without names or comments; labels and parameter names are numbered)
END_ORGANIZATION_BLOCK

ORGANIZATION_BLOCK "OBNL_FLT"	// OB 85
AUTHOR : Kamillas
VERSION : 0.1
BEGIN
// (block stored without names or comments; labels and parameter names are numbered)
END_ORGANIZATION_BLOCK

ORGANIZATION_BLOCK "RACK_FLT"	// OB 86
AUTHOR : Kamillas
VERSION : 0.1
BEGIN
// (block stored without names or comments; labels and parameter names are numbered)
END_ORGANIZATION_BLOCK

ORGANIZATION_BLOCK "PROG_ERR"	// OB 121
AUTHOR : Kamillas
VERSION : 0.1
BEGIN
// (block stored without names or comments; labels and parameter names are numbered)
END_ORGANIZATION_BLOCK

ORGANIZATION_BLOCK "MOD_ERR"	// OB 122
AUTHOR : Kamillas
VERSION : 0.1
BEGIN
// (block stored without names or comments; labels and parameter names are numbered)
END_ORGANIZATION_BLOCK
